C01878=0.000,57.118,70.285,-147.5034,-0.0009,0.0000
C01879=0.000,55.957,72.154,-148.8002,-0.0009,0.0000
C01880=1.768,55.936,72.129,-148.8075,-1.3174,0.0000
C01881=4.219,55.892,72.166,-149.9044,3.8027,0.0000
C01882=7.293,56.844,73.015,-167.6227,12.5357,0.0000
C01883=8.627,60.270,75.143,179.6232,-2.0390,0.0000
C01884=9.417,65.995,78.036,179.4118,-3.7953,0.0000
C01885=10.308,73.408,80.927,179.3669,-4.3506,0.0000
C01886=11.295,81.446,83.062,179.3315,-4.6371,0.0000
C01887=12.427,88.723,84.088,178.6153,-4.2623,0.0000
C01888=15.989,94.030,84.621,177.8322,-1.8057,0.0000
C01889=21.612,96.617,85.050,178.6701,-0.2203,0.0000
C01890=28.131,95.953,85.481,179.9155,0.0246,0.0000
C01891=34.883,93.717,85.762,179.9905,0.0035,0.0000
C01892=41.602,90.934,85.762,179.9908,0.0042,0.0000
C01893=47.957,87.741,85.481,179.9228,0.0423,0.0000
C01894=53.037,83.601,85.050,179.2153,1.0961,0.0000
C01895=55.184,77.795,84.621,179.7437,2.8086,0.0000
C01896=53.949,71.524,84.088,-177.9607,3.9923,0.0000
C01897=49.604,65.578,83.062,-177.1889,3.7534,0.0000
C01898=44.618,59.196,80.927,-177.3673,3.5255,0.0000
C01899=40.007,53.324,78.036,-177.7295,3.1005,0.0000
C01900=36.517,48.718,75.143,-178.8242,1.7083,0.0000
C01901=35.037,45.351,73.015,179.8825,-17.3486,0.0000
C01902=36.538,42.505,72.166,-160.0580,-24.5520,0.0000
C01903=38.303,40.803,72.129,-156.0408,-22.3844,0.0000
C01904=39.567,39.567,72.154,-156.8171,-23.1818,0.0000
C01905=40.803,38.303,72.129,-157.6162,-23.9597,0.0000
C01906=42.506,36.538,72.166,-155.4471,-19.9396,0.0000
C01907=45.352,35.037,73.015,-162.6519,0.1179,0.0000
C01908=48.718,36.517,75.143,178.2917,-1.1758,0.0000
C01909=53.324,40.007,78.036,176.8995,-2.2705,0.0000
C01910=59.196,44.618,80.927,176.4745,-2.6327,0.0000
C01911=65.578,49.604,83.062,176.2466,-2.8111,0.0000
C01912=71.524,53.949,84.088,176.0077,-2.0393,0.0000
C01913=77.795,55.184,84.621,177.1914,0.2563,0.0000
C01914=83.601,53.037,85.050,178.9039,0.7847,0.0000
C01915=87.741,47.957,85.481,179.9577,0.0772,0.0000
C01916=90.934,41.602,85.762,179.9958,0.0092,0.0000
C01917=93.717,34.883,85.762,179.9965,0.0095,0.0000
C01918=95.953,28.131,85.481,179.9754,0.0845,0.0000
C01919=96.617,21.612,85.050,-179.7797,1.3299,0.0000
C01920=94.030,15.989,84.621,-178.1943,2.1678,0.0000
C01921=88.723,12.427,84.088,-175.7377,1.3847,0.0000
C01922=81.446,11.295,83.062,-175.3629,0.6685,0.0000
C01923=73.408,10.308,80.927,-175.6494,0.6331,0.0000
C01924=65.995,9.417,78.036,-176.2047,0.5882,0.0000
C01925=60.270,8.627,75.143,-177.9610,0.3768,0.0000
C01926=56.844,7.293,73.015,167.4643,-12.3773,0.0000
C01927=55.892,4.219,72.166,176.1973,-30.0956,0.0000
C01928=55.936,1.768,72.129,-178.6826,-31.1925,0.0000
C01929=55.957,0.000,72.154,-179.9991,-31.1998,0.0000
C01930=55.936,-1.767,72.129,178.6816,-31.1926,0.0000
C01931=55.892,-4.220,72.166,-176.1946,-30.0948,0.0000
C01932=56.844,-7.293,73.015,-167.4645,-12.3766,0.0000
C01933=60.270,-8.627,75.143,177.9610,0.3768,0.0000
C01934=65.995,-9.417,78.036,176.2047,0.5882,0.0000
C01935=73.408,-10.308,80.927,175.6494,0.6331,0.0000
C01936=81.446,-11.295,83.062,175.3629,0.6685,0.0000
C01937=88.723,-12.427,84.088,175.7377,1.3847,0.0000
C01938=94.030,-15.989,84.621,178.1943,2.1678,0.0000
C01939=96.617,-21.612,85.050,179.7797,1.3299,0.0000
C01940=95.953,-28.131,85.481,-179.9754,0.0845,0.0000
C01941=93.717,-34.883,85.762,-179.9965,0.0095,0.0000
C01942=90.934,-41.602,85.762,-179.9958,0.0092,0.0000
C01943=87.741,-47.957,85.481,-179.9577,0.0772,0.0000
C01944=83.601,-53.037,85.050,-178.9039,0.7847,0.0000
C01945=77.795,-55.184,84.621,-177.1914,0.2563,0.0000
C01946=71.524,-53.949,84.088,-176.0077,-2.0393,0.0000
C01947=65.578,-49.604,83.062,-176.2466,-2.8111,0.0000
C01948=59.196,-44.618,80.927,-176.4745,-2.6327,0.0000
C01949=53.324,-40.007,78.036,-176.8995,-2.2705,0.0000
C01950=48.718,-36.517,75.143,-178.2917,-1.1758,0.0000
C01951=45.351,-35.037,73.015,162.6514,0.1175,0.0000
C01952=42.505,-36.538,72.166,155.4480,-19.9420,0.0000
C01953=40.803,-38.303,72.129,157.6156,-23.9592,0.0000
C01954=39.567,-39.567,72.154,156.8182,-23.1829,0.0000
C01955=38.303,-40.803,72.129,156.0403,-22.3838,0.0000
C01956=36.538,-42.506,72.166,160.0604,-24.5529,0.0000
C01957=35.037,-45.352,73.015,-179.8821,-17.3481,0.0000
C01958=36.517,-48.718,75.143,178.8242,1.7083,0.0000
C01959=40.007,-53.324,78.036,177.7295,3.1005,0.0000
C01960=44.618,-59.196,80.927,177.3673,3.5255,0.0000
C01961=49.604,-65.578,83.062,177.1889,3.7534,0.0000
C01962=53.949,-71.524,84.088,177.9607,3.9923,0.0000
C01963=55.184,-77.795,84.621,-179.7437,2.8086,0.0000
C01964=53.037,-83.601,85.050,-179.2153,1.0961,0.0000
C01965=47.957,-87.741,85.481,-179.9228,0.0423,0.0000
C01966=41.602,-90.934,85.762,-179.9908,0.0042,0.0000
C01967=34.883,-93.717,85.762,-179.9905,0.0035,0.0000
C01968=28.131,-95.953,85.481,-179.9155,0.0246,0.0000
C01969=21.612,-96.617,85.050,-178.6701,-0.2203,0.0000
C01970=15.989,-94.030,84.621,-177.8322,-1.8057,0.0000
C01971=12.427,-88.723,84.088,-178.6153,-4.2623,0.0000
C01972=11.295,-81.446,83.062,-179.3315,-4.6371,0.0000
C01973=10.308,-73.408,80.927,-179.3669,-4.3506,0.0000
C01974=9.417,-65.995,78.036,-179.4118,-3.7953,0.0000
C01975=8.627,-60.270,75.143,-179.6232,-2.0390,0.0000
C01976=7.293,-56.844,73.015,167.6227,12.5357,0.0000
C01977=4.219,-55.892,72.166,149.9044,3.8027,0.0000
C01978=1.768,-55.936,72.129,148.8075,-1.3174,0.0000
C01979=0.000,-55.957,72.154,148.8002,-0.0009,0.0000
C01980=0.000,-55.957,72.154,148.8002,-0.0009,0.0000
C01981=-1.767,-55.936,72.129,148.8074,1.3184,0.0000
C01982=-4.220,-55.892,72.166,149.9052,-3.8054,0.0000
C01983=-7.293,-56.844,73.015,167.6234,-12.5355,0.0000
C01984=-8.627,-60.270,75.143,-179.6232,2.0390,0.0000
C01985=-9.417,-65.995,78.036,-179.4118,3.7953,0.0000
C01986=-10.308,-73.408,80.927,-179.3669,4.3506,0.0000
C01987=-11.295,-81.446,83.062,-179.3315,4.6371,0.0000
C01988=-12.427,-88.723,84.088,-178.6153,4.2623,0.0000
C01989=-15.989,-94.030,84.621,-177.8322,1.8057,0.0000
C01990=-21.612,-96.617,85.050,-178.6701,0.2203,0.0000
C01991=-28.131,-95.953,85.481,-179.9155,-0.0246,0.0000
C01992=-34.883,-93.717,85.762,-179.9905,-0.0035,0.0000
C01993=-41.602,-90.934,85.762,-179.9908,-0.0042,0.0000
C01994=-47.957,-87.741,85.481,-179.9228,-0.0423,0.0000
C01995=-53.037,-83.601,85.050,-179.2153,-1.0961,0.0000
C01996=-55.184,-77.795,84.621,-179.7437,-2.8086,0.0000
C01997=-53.949,-71.524,84.088,177.9607,-3.9923,0.0000
C01998=-49.604,-65.578,83.062,177.1889,-3.7534,0.0000
C01999=-44.618,-59.196,80.927,177.3673,-3.5255,0.0000
///TOOL 0
///POSTYPE ANGLE
///ANGLE
EC00000=-104.1038,0.0000
EC00001=-101.5206,0.0000
EC00002=-99.9757,0.0000
EC00003=-99.7146,0.0000
EC00004=-99.6525,0.0000
EC00005=-99.5501,0.0000
EC00006=-99.1897,0.0000
EC00007=-97.9963,0.0000
EC00008=-95.1629,0.0000
EC00009=-92.4517,0.0000
EC00010=-90.0000,0.0000
EC00011=-87.5483,0.0000
EC00012=-84.8371,0.0000
EC00013=-82.0037,0.0000
EC00014=-80.8103,0.0000
EC00015=-80.4499,0.0000
EC00016=-80.3475,0.0000
EC00017=-80.2854,0.0000
EC00018=-80.0243,0.0000
EC00019=-78.4794,0.0000
EC00020=-75.8962,0.0000
EC00021=-72.7026,0.0000
EC00022=-69.2567,0.0000
EC00023=-65.7434,0.0000
EC00024=-62.2974,0.0000
EC00025=-59.1038,0.0000
EC00026=-56.5207,0.0000
EC00027=-54.9755,0.0000
EC00028=-54.7145,0.0000
EC00029=-54.6524,0.0000
EC00030=-54.5505,0.0000
EC00031=-54.1895,0.0000
EC00032=-52.9962,0.0000
EC00033=-50.1628,0.0000
EC00034=-47.4518,0.0000
EC00035=-45.0000,0.0000
EC00036=-42.5482,0.0000
EC00037=-39.8372,0.0000
EC00038=-37.0034,0.0000
EC00039=-35.8105,0.0000
EC00040=-35.4495,0.0000
EC00041=-35.3476,0.0000
EC00042=-35.2855,0.0000
EC00043=-35.0245,0.0000
EC00044=-33.4793,0.0000
EC00045=-30.8962,0.0000
EC00046=-27.7026,0.0000
EC00047=-24.2566,0.0000
EC00048=-20.7433,0.0000
EC00049=-17.2974,0.0000
EC00050=-14.1038,0.0000
EC00051=-11.5206,0.0000
EC00052=-9.9757,0.0000
EC00053=-9.7146,0.0000
EC00054=-9.6525,0.0000
EC00055=-9.5501,0.0000
EC00056=-9.1897,0.0000
EC00057=-7.9963,0.0000
EC00058=-5.1629,0.0000
EC00059=-2.4517,0.0000
EC00060=0.0000,0.0000
EC00061=0.0000,0.0000
EC00062=2.3954,0.0000
EC00063=5.0881,0.0000
EC00064=7.9350,0.0000
EC00065=9.0911,0.0000
EC00066=9.4060,0.0000
EC00067=9.4709,0.0000
EC00068=9.5004,0.0000
EC00069=9.7298,0.0000
EC00070=11.2851,0.0000
EC00071=13.9122,0.0000
EC00072=17.1736,0.0000
EC00073=20.7008,0.0000
EC00074=24.2992,0.0000
EC00075=27.8267,0.0000
EC00076=31.0877,0.0000
EC00077=33.7152,0.0000
EC00078=35.2699,0.0000
EC00079=35.4993,0.0000
EC00080=35.5293,0.0000
EC00081=35.5938,0.0000
EC00082=35.9087,0.0000
EC00083=37.0654,0.0000
EC00084=39.9123,0.0000
EC00085=42.6047,0.0000
EC00086=45.0000,0.0000
EC00087=47.3953,0.0000
EC00088=50.0883,0.0000
EC00089=52.9346,0.0000
EC00090=54.0913,0.0000
EC00091=54.4062,0.0000
EC00092=54.4707,0.0000
EC00093=54.5007,0.0000
EC00094=54.7301,0.0000
EC00095=56.2848,0.0000
EC00096=58.9123,0.0000
EC00097=62.1733,0.0000
EC00098=65.7008,0.0000
EC00099=69.2992,0.0000
EC00100=72.8264,0.0000
EC00101=76.0878,0.0000
EC00102=78.7149,0.0000
EC00103=80.2702,0.0000
EC00104=80.4996,0.0000
EC00105=80.5291,0.0000
EC00106=80.5940,0.0000
EC00107=80.9089,0.0000
EC00108=82.0650,0.0000
EC00109=84.9119,0.0000
EC00110=87.6046,0.0000
EC00111=90.0000,0.0000
EC00112=92.3954,0.0000
EC00113=95.0881,0.0000
EC00114=97.9350,0.0000
EC00115=99.0911,0.0000
EC00116=99.4060,0.0000
EC00117=99.4709,0.0000
EC00118=99.5004,0.0000
EC00119=99.7298,0.0000
EC00120=101.2851,0.0000
EC00121=103.9122,0.0000
EC00122=107.1736,0.0000
EC00123=110.7008,0.0000
EC00124=114.2992,0.0000
EC00125=117.8267,0.0000
EC00126=121.0877,0.0000
EC00127=123.7152,0.0000
EC00128=125.2699,0.0000
EC00129=125.4993,0.0000
EC00130=125.5293,0.0000
EC00131=125.5938,0.0000
EC00132=125.9087,0.0000
EC00133=127.0654,0.0000
EC00134=129.9123,0.0000
EC00135=132.6047,0.0000
EC00136=135.0000,0.0000
EC00137=137.3953,0.0000
EC00138=140.0883,0.0000
EC00139=142.9346,0.0000
EC00140=144.0913,0.0000
EC00141=144.4062,0.0000
EC00142=144.4707,0.0000
EC00143=144.5007,0.0000
EC00144=144.7301,0.0000
EC00145=146.2848,0.0000
EC00146=148.9123,0.0000
EC00147=152.1733,0.0000
EC00148=155.7008,0.0000
EC00149=159.2992,0.0000
EC00150=162.8264,0.0000
EC00151=166.0878,0.0000
EC00152=168.7149,0.0000
EC00153=170.2702,0.0000
EC00154=170.4996,0.0000
EC00155=170.5291,0.0000
EC00156=170.5940,0.0000
EC00157=170.9089,0.0000
EC00158=172.0650,0.0000
EC00159=174.9119,0.0000
EC00160=177.6046,0.0000
EC00161=180.0000,0.0000
EC00162=180.0000,0.0000
EC00163=-177.6046,0.0000
EC00164=-174.9119,0.0000
EC00165=-172.0650,0.0000
EC00166=-170.9089,0.0000
EC00167=-170.5940,0.0000
EC00168=-170.5291,0.0000
EC00169=-170.4996,0.0000
EC00170=-170.2702,0.0000
EC00171=-168.7149,0.0000
EC00172=-166.0878,0.0000
EC00173=-162.8264,0.0000
EC00174=-159.2992,0.0000
EC00175=-155.7008,0.0000
EC00176=-152.1733,0.0000
EC00177=-148.9123,0.0000
EC00178=-146.2848,0.0000
EC00179=-144.7301,0.0000
EC00180=-144.5007,0.0000
EC00181=-144.4707,0.0000
EC00182=-144.4062,0.0000
EC00183=-144.0913,0.0000
EC00184=-142.9346,0.0000
EC00185=-140.0877,0.0000
EC00186=-137.3953,0.0000
EC00187=-135.0000,0.0000
EC00188=-132.6047,0.0000
EC00189=-129.9117,0.0000
EC00190=-127.0654,0.0000
EC00191=-125.9087,0.0000
EC00192=-125.5938,0.0000
EC00193=-125.5293,0.0000
EC00194=-125.4993,0.0000
EC00195=-125.2699,0.0000
EC00196=-123.7152,0.0000
EC00197=-121.0877,0.0000
EC00198=-117.8267,0.0000
EC00199=-114.2992,0.0000
EC00200=-110.7008,0.0000
EC00201=-107.1736,0.0000
EC00202=-103.9122,0.0000
EC00203=-101.2851,0.0000
EC00204=-99.7298,0.0000
EC00205=-99.5004,0.0000
EC00206=-99.4709,0.0000
EC00207=-99.4060,0.0000
EC00208=-99.0911,0.0000
EC00209=-97.9350,0.0000
EC00210=-95.0881,0.0000
EC00211=-92.3954,0.0000
EC00212=-90.0000,0.0000
EC00213=-87.6046,0.0000
EC00214=-84.9119,0.0000
EC00215=-82.0650,0.0000
EC00216=-80.9089,0.0000
EC00217=-80.5940,0.0000
EC00218=-80.5291,0.0000
EC00219=-80.4996,0.0000
EC00220=-80.2702,0.0000
EC00221=-78.7149,0.0000
EC00222=-76.0878,0.0000
EC00223=-72.8264,0.0000
EC00224=-69.2992,0.0000
EC00225=-65.7008,0.0000
EC00226=-62.1733,0.0000
EC00227=-58.9123,0.0000
EC00228=-56.2848,0.0000
EC00229=-54.7301,0.0000
EC00230=-54.5007,0.0000
EC00231=-54.4707,0.0000
EC00232=-54.4062,0.0000
EC00233=-54.0913,0.0000
EC00234=-52.9346,0.0000
EC00235=-50.0877,0.0000
EC00236=-47.3953,0.0000
EC00237=-45.0000,0.0000
EC00238=-42.6047,0.0000
EC00239=-39.9117,0.0000
EC00240=-37.0654,0.0000
EC00241=-35.9087,0.0000
EC00242=-35.5938,0.0000
EC00243=-35.5293,0.0000
EC00244=-35.4993,0.0000
EC00245=-35.2699,0.0000
EC00246=-33.7152,0.0000
EC00247=-31.0877,0.0000
EC00248=-27.8267,0.0000
EC00249=-24.2992,0.0000
EC00250=-20.7008,0.0000
EC00251=-17.1736,0.0000
EC00252=-13.9122,0.0000
EC00253=-11.2851,0.0000
EC00254=-9.7298,0.0000
EC00255=-9.5004,0.0000
EC00256=-9.4709,0.0000
EC00257=-9.4060,0.0000
EC00258=-9.0911,0.0000
EC00259=-7.9350,0.0000
EC00260=-5.0881,0.0000
EC00261=-2.3954,0.0000
EC00262=0.0000,0.0000
EC00263=0.0000,0.0000
EC00264=2.3363,0.0000
EC00265=5.0104,0.0000
EC00266=7.8714,0.0000
EC00267=8.9912,0.0000
EC00268=9.2604,0.0000
EC00269=9.2892,0.0000
EC00270=9.2905,0.0000
EC00271=9.4907,0.0000
EC00272=11.0568,0.0000
EC00273=13.7273,0.0000
EC00274=17.0541,0.0000
EC00275=20.6599,0.0000
EC00276=24.3400,0.0000
EC00277=27.9461,0.0000
EC00278=31.2727,0.0000
EC00279=33.9430,0.0000
EC00280=35.5096,0.0000
EC00281=35.7099,0.0000
EC00282=35.7103,0.0000
EC00283=35.7399,0.0000
EC00284=36.0092,0.0000
EC00285=37.1289,0.0000
EC00286=39.9895,0.0000
EC00287=42.6632,0.0000
EC00288=45.0000,0.0000
EC00289=47.3362,0.0000
EC00290=50.0105,0.0000
EC00291=52.8711,0.0000
EC00292=53.9908,0.0000
EC00293=54.2601,0.0000
EC00294=54.2897,0.0000
EC00295=54.2901,0.0000
EC00296=54.4904,0.0000
EC00297=56.0570,0.0000
EC00298=58.7273,0.0000
EC00299=62.0539,0.0000
EC00300=65.6600,0.0000
EC00301=69.3401,0.0000
EC00302=72.9459,0.0000
EC00303=76.2727,0.0000
EC00304=78.9432,0.0000
EC00305=80.5093,0.0000
EC00306=80.7095,0.0000
EC00307=80.7108,0.0000
EC00308=80.7396,0.0000
EC00309=81.0088,0.0000
EC00310=82.1286,0.0000
EC00311=84.9896,0.0000
EC00312=87.6637,0.0000
EC00313=90.0000,0.0000
EC00314=92.3363,0.0000
EC00315=95.0112,0.0000
EC00316=97.8714,0.0000
EC00317=98.9912,0.0000
EC00318=99.2604,0.0000
EC00319=99.2892,0.0000
EC00320=99.2905,0.0000
EC00321=99.4907,0.0000
EC00322=101.0568,0.0000
EC00323=103.7273,0.0000
EC00324=107.0541,0.0000
EC00325=110.6599,0.0000
EC00326=114.3400,0.0000
EC00327=117.9461,0.0000
EC00328=121.2727,0.0000
EC00329=123.9430,0.0000
EC00330=125.5096,0.0000
EC00331=125.7099,0.0000
EC00332=125.7103,0.0000
EC00333=125.7399,0.0000
EC00334=126.0092,0.0000
EC00335=127.1289,0.0000
EC00336=129.9895,0.0000
EC00337=132.6632,0.0000
EC00338=135.0000,0.0000
EC00339=137.3362,0.0000
EC00340=140.0105,0.0000
EC00341=142.8711,0.0000
EC00342=143.9908,0.0000
EC00343=144.2601,0.0000
EC00344=144.2897,0.0000
EC00345=144.2901,0.0000
EC00346=144.4904,0.0000
EC00347=146.0570,0.0000
EC00348=148.7273,0.0000
EC00349=152.0539,0.0000
EC00350=155.6600,0.0000
EC00351=159.3401,0.0000
EC00352=162.9459,0.0000
EC00353=166.2727,0.0000
EC00354=168.9432,0.0000
EC00355=170.5093,0.0000
EC00356=170.7095,0.0000
EC00357=170.7108,0.0000
EC00358=170.7396,0.0000
EC00359=171.0088,0.0000
EC00360=172.1286,0.0000
EC00361=174.9896,0.0000
EC00362=177.6637,0.0000
EC00363=180.0000,0.0000
EC00364=180.0000,0.0000
EC00365=-177.6637,0.0000
EC00366=-174.9888,0.0000
EC00367=-172.1286,0.0000
EC00368=-171.0088,0.0000
EC00369=-170.7396,0.0000
EC00370=-170.7108,0.0000
EC00371=-170.7095,0.0000
EC00372=-170.5093,0.0000
EC00373=-168.9432,0.0000
EC00374=-166.2727,0.0000
EC00375=-162.9459,0.0000
EC00376=-159.3401,0.0000
EC00377=-155.6600,0.0000
EC00378=-152.0539,0.0000
EC00379=-148.7273,0.0000
EC00380=-146.0570,0.0000
EC00381=-144.4904,0.0000
EC00382=-144.2901,0.0000
EC00383=-144.2897,0.0000
EC00384=-144.2601,0.0000
EC00385=-143.9908,0.0000
EC00386=-142.8711,0.0000
EC00387=-140.0105,0.0000
EC00388=-137.3368,0.0000
EC00389=-135.0000,0.0000
EC00390=-132.6638,0.0000
EC00391=-129.9895,0.0000
EC00392=-127.1289,0.0000
EC00393=-126.0092,0.0000
EC00394=-125.7399,0.0000
EC00395=-125.7103,0.0000
EC00396=-125.7099,0.0000
EC00397=-125.5096,0.0000
EC00398=-123.9430,0.0000
EC00399=-121.2727,0.0000
EC00400=-117.9461,0.0000
EC00401=-114.3400,0.0000
EC00402=-110.6599,0.0000
EC00403=-107.0541,0.0000
EC00404=-103.7273,0.0000
EC00405=-101.0568,0.0000
EC00406=-99.4907,0.0000
EC00407=-99.2905,0.0000
EC00408=-99.2892,0.0000
EC00409=-99.2604,0.0000
EC00410=-98.9912,0.0000
EC00411=-97.8714,0.0000
EC00412=-95.0104,0.0000
EC00413=-92.3363,0.0000
EC00414=-90.0000,0.0000
EC00415=-87.6637,0.0000
EC00416=-84.9888,0.0000
EC00417=-82.1286,0.0000
EC00418=-81.0088,0.0000
EC00419=-80.7396,0.0000
EC00420=-80.7108,0.0000
EC00421=-80.7095,0.0000
EC00422=-80.5093,0.0000
EC00423=-78.9432,0.0000
EC00424=-76.2727,0.0000
EC00425=-72.9459,0.0000
EC00426=-69.3401,0.0000
EC00427=-65.6600,0.0000
EC00428=-62.0539,0.0000
EC00429=-58.7273,0.0000
EC00430=-56.0570,0.0000
EC00431=-54.4904,0.0000
EC00432=-54.2901,0.0000
EC00433=-54.2897,0.0000
EC00434=-54.2601,0.0000
EC00435=-53.9908,0.0000
EC00436=-52.8711,0.0000
EC00437=-50.0105,0.0000
EC00438=-47.3368,0.0000
EC00439=-45.0000,0.0000
EC00440=-42.6638,0.0000
EC00441=-39.9895,0.0000
EC00442=-37.1289,0.0000
EC00443=-36.0092,0.0000
EC00444=-35.7399,0.0000
EC00445=-35.7103,0.0000
EC00446=-35.7099,0.0000
EC00447=-35.5096,0.0000
EC00448=-33.9430,0.0000
EC00449=-31.2727,0.0000
EC00450=-27.9461,0.0000
EC00451=-24.3400,0.0000
EC00452=-20.6599,0.0000
EC00453=-17.0541,0.0000
EC00454=-13.7273,0.0000
EC00455=-11.0568,0.0000
EC00456=-9.4907,0.0000
EC00457=-9.2905,0.0000
EC00458=-9.2892,0.0000
EC00459=-9.2604,0.0000
EC00460=-8.9912,0.0000
EC00461=-7.8714,0.0000
EC00462=-5.0112,0.0000
EC00463=-2.3363,0.0000
EC00464=0.0000,0.0000
EC00465=0.0000,0.0000
EC00466=2.2761,0.0000
EC00467=4.9310,0.0000
EC00468=7.8063,0.0000
EC00469=8.8881,0.0000
EC00470=9.1126,0.0000
EC00471=9.1102,0.0000
EC00472=9.0849,0.0000
EC00473=9.2589,0.0000
EC00474=10.8371,0.0000
EC00475=13.5503,0.0000
EC00476=16.9400,0.0000
EC00477=20.6205,0.0000
EC00478=24.3795,0.0000
EC00479=28.0601,0.0000
EC00480=31.4498,0.0000
EC00481=34.1627,0.0000
EC00482=35.7411,0.0000
EC00483=35.9150,0.0000
EC00484=35.8901,0.0000
EC00485=35.8871,0.0000
EC00486=36.1114,0.0000
EC00487=37.1942,0.0000
EC00488=40.0690,0.0000
EC00489=42.7235,0.0000
EC00490=45.0000,0.0000
EC00491=47.2759,0.0000
EC00492=49.9310,0.0000
EC00493=52.8058,0.0000
EC00494=53.8886,0.0000
EC00495=54.1129,0.0000
EC00496=54.1099,0.0000
EC00497=54.0850,0.0000
EC00498=54.2589,0.0000
EC00499=55.8373,0.0000
EC00500=58.5502,0.0000
EC00501=61.9399,0.0000
EC00502=65.6205,0.0000
EC00503=69.3795,0.0000
EC00504=73.0600,0.0000
EC00505=76.4497,0.0000
EC00506=79.1629,0.0000
EC00507=80.7411,0.0000
EC00508=80.9151,0.0000
EC00509=80.8898,0.0000
EC00510=80.8874,0.0000
EC00511=81.1119,0.0000
EC00512=82.1937,0.0000
EC00513=85.0690,0.0000
EC00514=87.7239,0.0000
EC00515=90.0000,0.0000
EC00516=92.2761,0.0000
EC00517=94.9310,0.0000
EC00518=97.8063,0.0000
EC00519=98.8881,0.0000
EC00520=99.1126,0.0000
EC00521=99.1102,0.0000
EC00522=99.0849,0.0000
EC00523=99.2589,0.0000
EC00524=100.8371,0.0000
EC00525=103.5503,0.0000
EC00526=106.9400,0.0000
EC00527=110.6205,0.0000
EC00528=114.3795,0.0000
EC00529=118.0601,0.0000
EC00530=121.4498,0.0000
EC00531=124.1627,0.0000
EC00532=125.7411,0.0000
EC00533=125.9150,0.0000
EC00534=125.8901,0.0000
EC00535=125.8871,0.0000
EC00536=126.1114,0.0000
EC00537=127.1942,0.0000
EC00538=130.0690,0.0000
EC00539=132.7235,0.0000
EC00540=135.0000,0.0000
EC00541=137.2759,0.0000
EC00542=139.9310,0.0000
EC00543=142.8058,0.0000
EC00544=143.8886,0.0000
EC00545=144.1129,0.0000
EC00546=144.1099,0.0000
EC00547=144.0850,0.0000
EC00548=144.2589,0.0000
EC00549=145.8373,0.0000
EC00550=148.5502,0.0000
EC00551=151.9399,0.0000
EC00552=155.6205,0.0000
EC00553=159.3795,0.0000
EC00554=163.0600,0.0000
EC00555=166.4497,0.0000
EC00556=169.1629,0.0000
EC00557=170.7411,0.0000
EC00558=170.9151,0.0000
EC00559=170.8898,0.0000
EC00560=170.8874,0.0000
EC00561=171.1119,0.0000
EC00562=172.1937,0.0000
EC00563=175.0690,0.0000
EC00564=177.7239,0.0000
EC00565=180.0000,0.0000
EC00566=180.0000,0.0000
EC00567=-177.7239,0.0000
EC00568=-175.0690,0.0000
EC00569=-172.1937,0.0000
EC00570=-171.1119,0.0000
EC00571=-170.8874,0.0000
EC00572=-170.8898,0.0000
EC00573=-170.9151,0.0000
EC00574=-170.7411,0.0000
EC00575=-169.1629,0.0000
EC00576=-166.4497,0.0000
EC00577=-163.0600,0.0000
EC00578=-159.3795,0.0000
EC00579=-155.6205,0.0000
EC00580=-151.9399,0.0000
EC00581=-148.5502,0.0000
EC00582=-145.8373,0.0000
EC00583=-144.2589,0.0000
EC00584=-144.0850,0.0000
EC00585=-144.1099,0.0000
EC00586=-144.1129,0.0000
EC00587=-143.8886,0.0000
EC00588=-142.8058,0.0000
EC00589=-139.9310,0.0000
EC00590=-137.2765,0.0000
EC00591=-135.0000,0.0000
EC00592=-132.7241,0.0000
EC00593=-130.0690,0.0000
EC00594=-127.1942,0.0000
EC00595=-126.1114,0.0000
EC00596=-125.8871,0.0000
EC00597=-125.8901,0.0000
EC00598=-125.9150,0.0000
EC00599=-125.7411,0.0000
EC00600=-124.1627,0.0000
EC00601=-121.4498,0.0000
EC00602=-118.0601,0.0000
EC00603=-114.3795,0.0000
EC00604=-110.6205,0.0000
EC00605=-106.9400,0.0000
EC00606=-103.5503,0.0000
EC00607=-100.8371,0.0000
EC00608=-99.2589,0.0000
EC00609=-99.0849,0.0000
EC00610=-99.1102,0.0000
EC00611=-99.1126,0.0000
EC00612=-98.8881,0.0000
EC00613=-97.8063,0.0000
EC00614=-94.9310,0.0000
EC00615=-92.2761,0.0000
EC00616=-90.0000,0.0000
EC00617=-87.7239,0.0000
EC00618=-85.0690,0.0000
EC00619=-82.1937,0.0000
EC00620=-81.1119,0.0000
EC00621=-80.8874,0.0000
EC00622=-80.8898,0.0000
EC00623=-80.9151,0.0000
EC00624=-80.7411,0.0000
EC00625=-79.1629,0.0000
EC00626=-76.4497,0.0000
EC00627=-73.0600,0.0000
EC00628=-69.3795,0.0000
EC00629=-65.6205,0.0000
EC00630=-61.9399,0.0000
EC00631=-58.5502,0.0000
EC00632=-55.8373,0.0000
EC00633=-54.2589,0.0000
EC00634=-54.0850,0.0000
EC00635=-54.1099,0.0000
EC00636=-54.1129,0.0000
EC00637=-53.8886,0.0000
EC00638=-52.8058,0.0000
EC00639=-49.9310,0.0000
EC00640=-47.2765,0.0000
EC00641=-45.0000,0.0000
EC00642=-42.7241,0.0000
EC00643=-40.0690,0.0000
EC00644=-37.1942,0.0000
EC00645=-36.1114,0.0000
EC00646=-35.8871,0.0000
EC00647=-35.8901,0.0000
EC00648=-35.9150,0.0000
EC00649=-35.7411,0.0000
EC00650=-34.1627,0.0000
EC00651=-31.4498,0.0000
EC00652=-28.0601,0.0000
EC00653=-24.3795,0.0000
EC00654=-20.6205,0.0000
EC00655=-16.9400,0.0000
EC00656=-13.5503,0.0000
EC00657=-10.8371,0.0000
EC00658=-9.2589,0.0000
EC00659=-9.0849,0.0000
EC00660=-9.1102,0.0000
EC00661=-9.1126,0.0000
EC00662=-8.8881,0.0000
EC00663=-7.8063,0.0000
EC00664=-4.9310,0.0000
EC00665=-2.2761,0.0000
EC00666=0.0000,0.0000
EC00667=0.0000,0.0000
EC00668=2.2137,0.0000
EC00669=4.8488,0.0000
EC00670=7.7390,0.0000
EC00671=8.7837,0.0000
EC00672=8.9651,0.0000
EC00673=8.9329,0.0000
EC00674=8.8862,0.0000
EC00675=9.0366,0.0000
EC00676=10.6278,0.0000
EC00677=13.3823,0.0000
EC00678=16.8314,0.0000
EC00679=20.5837,0.0000
EC00680=24.4165,0.0000
EC00681=28.1685,0.0000
EC00682=31.6178,0.0000
EC00683=34.3719,0.0000
EC00684=35.9638,0.0000
EC00685=36.1137,0.0000
EC00686=36.0668,0.0000
EC00687=36.0347,0.0000
EC00688=36.2163,0.0000
EC00689=37.2611,0.0000
EC00690=40.1513,0.0000
EC00691=42.7862,0.0000
EC00692=45.0000,0.0000
EC00693=47.2138,0.0000
EC00694=49.8487,0.0000
EC00695=52.7389,0.0000
EC00696=53.7837,0.0000
EC00697=53.9653,0.0000
EC00698=53.9332,0.0000
EC00699=53.8863,0.0000
EC00700=54.0362,0.0000
EC00701=55.6281,0.0000
EC00702=58.3822,0.0000
EC00703=61.8315,0.0000
EC00704=65.5835,0.0000
EC00705=69.4163,0.0000
EC00706=73.1686,0.0000
EC00707=76.6177,0.0000
EC00708=79.3722,0.0000
EC00709=80.9634,0.0000
EC00710=81.1138,0.0000
EC00711=81.0671,0.0000
EC00712=81.0349,0.0000
EC00713=81.2163,0.0000
EC00714=82.2610,0.0000
EC00715=85.1512,0.0000
EC00716=87.7863,0.0000
EC00717=90.0000,0.0000
EC00718=92.2137,0.0000
EC00719=94.8488,0.0000
EC00720=97.7390,0.0000
EC00721=98.7837,0.0000
EC00722=98.9651,0.0000
EC00723=98.9329,0.0000
EC00724=98.8862,0.0000
EC00725=99.0366,0.0000
EC00726=100.6278,0.0000
EC00727=103.3823,0.0000
EC00728=106.8314,0.0000
EC00729=110.5837,0.0000
EC00730=114.4165,0.0000
EC00731=118.1685,0.0000
EC00732=121.6178,0.0000
EC00733=124.3719,0.0000
EC00734=125.9638,0.0000
EC00735=126.1137,0.0000
EC00736=126.0668,0.0000
EC00737=126.0347,0.0000
EC00738=126.2163,0.0000
EC00739=127.2611,0.0000
EC00740=130.1513,0.0000
EC00741=132.7862,0.0000
EC00742=135.0000,0.0000
EC00743=137.2138,0.0000
EC00744=139.8487,0.0000
EC00745=142.7389,0.0000
EC00746=143.7837,0.0000
EC00747=143.9653,0.0000
EC00748=143.9332,0.0000
EC00749=143.8863,0.0000
EC00750=144.0362,0.0000
EC00751=145.6281,0.0000
EC00752=148.3822,0.0000
EC00753=151.8315,0.0000
EC00754=155.5835,0.0000
EC00755=159.4163,0.0000
EC00756=163.1686,0.0000
EC00757=166.6177,0.0000
EC00758=169.3722,0.0000
EC00759=170.9634,0.0000
EC00760=171.1138,0.0000
EC00761=171.0671,0.0000
EC00762=171.0349,0.0000
EC00763=171.2163,0.0000
EC00764=172.2610,0.0000
EC00765=175.1512,0.0000
EC00766=177.7863,0.0000
EC00767=180.0000,0.0000
EC00768=180.0000,0.0000
EC00769=-177.7863,0.0000
EC00770=-175.1512,0.0000
EC00771=-172.2610,0.0000
EC00772=-171.2163,0.0000
EC00773=-171.0349,0.0000
EC00774=-171.0671,0.0000
EC00775=-171.1138,0.0000
EC00776=-170.9634,0.0000
EC00777=-169.3722,0.0000
EC00778=-166.6177,0.0000
EC00779=-163.1686,0.0000
EC00780=-159.4163,0.0000
EC00781=-155.5835,0.0000
EC00782=-151.8315,0.0000
EC00783=-148.3822,0.0000
EC00784=-145.6281,0.0000
EC00785=-144.0362,0.0000
EC00786=-143.8863,0.0000
EC00787=-143.9332,0.0000
EC00788=-143.9653,0.0000
EC00789=-143.7837,0.0000
EC00790=-142.7389,0.0000
EC00791=-139.8487,0.0000
EC00792=-137.2138,0.0000
EC00793=-135.0000,0.0000
EC00794=-132.7862,0.0000
EC00795=-130.1513,0.0000
EC00796=-127.2611,0.0000
EC00797=-126.2163,0.0000
EC00798=-126.0347,0.0000
EC00799=-126.0668,0.0000
EC00800=-126.1137,0.0000
EC00801=-125.9638,0.0000
EC00802=-124.3719,0.0000
EC00803=-121.6178,0.0000
EC00804=-118.1685,0.0000
EC00805=-114.4165,0.0000
EC00806=-110.5837,0.0000
EC00807=-106.8314,0.0000
EC00808=-103.3823,0.0000
EC00809=-100.6278,0.0000
EC00810=-99.0366,0.0000
EC00811=-98.8862,0.0000
EC00812=-98.9329,0.0000
EC00813=-98.9651,0.0000
EC00814=-98.7837,0.0000
EC00815=-97.7390,0.0000
EC00816=-94.8488,0.0000
EC00817=-92.2137,0.0000
EC00818=-90.0000,0.0000
EC00819=-87.7863,0.0000
EC00820=-85.1512,0.0000
EC00821=-82.2610,0.0000
EC00822=-81.2163,0.0000
EC00823=-81.0349,0.0000
EC00824=-81.0671,0.0000
EC00825=-81.1138,0.0000
EC00826=-80.9634,0.0000
EC00827=-79.3722,0.0000
EC00828=-76.6177,0.0000
EC00829=-73.1686,0.0000
EC00830=-69.4163,0.0000
EC00831=-65.5835,0.0000
EC00832=-61.8315,0.0000
EC00833=-58.3822,0.0000
EC00834=-55.6281,0.0000
EC00835=-54.0362,0.0000
EC00836=-53.8863,0.0000
EC00837=-53.9332,0.0000
EC00838=-53.9653,0.0000
EC00839=-53.7837,0.0000
EC00840=-52.7389,0.0000
EC00841=-49.8487,0.0000
EC00842=-47.2138,0.0000
EC00843=-45.0000,0.0000
EC00844=-42.7862,0.0000
EC00845=-40.1513,0.0000
EC00846=-37.2611,0.0000
EC00847=-36.2163,0.0000
EC00848=-36.0347,0.0000
EC00849=-36.0668,0.0000
EC00850=-36.1137,0.0000
EC00851=-35.9638,0.0000
EC00852=-34.3719,0.0000
EC00853=-31.6178,0.0000
EC00854=-28.1685,0.0000
EC00855=-24.4165,0.0000
EC00856=-20.5837,0.0000
EC00857=-16.8314,0.0000
EC00858=-13.3823,0.0000
EC00859=-10.6278,0.0000
EC00860=-9.0366,0.0000
EC00861=-8.8862,0.0000
EC00862=-8.9329,0.0000
EC00863=-8.9651,0.0000
EC00864=-8.7837,0.0000
EC00865=-7.7390,0.0000
EC00866=-4.8488,0.0000
EC00867=-2.2137,0.0000
EC00868=0.0000,0.0000
EC00869=0.0000,0.0000
EC00870=2.1497,0.0000
EC00871=4.7644,0.0000
EC00872=7.6702,0.0000
EC00873=8.6786,0.0000
EC00874=8.8182,0.0000
EC00875=8.7594,0.0000
EC00876=8.6938,0.0000
EC00877=8.8243,0.0000
EC00878=10.4296,0.0000
EC00879=13.2238,0.0000
EC00880=16.7302,0.0000
EC00881=20.5487,0.0000
EC00882=24.4516,0.0000
EC00883=28.2700,0.0000
EC00884=31.7764,0.0000
EC00885=34.5698,0.0000
EC00886=36.1755,0.0000
EC00887=36.3059,0.0000
EC00888=36.2401,0.0000
EC00889=36.1817,0.0000
EC00890=36.3218,0.0000
EC00891=37.3300,0.0000
EC00892=40.2352,0.0000
EC00893=42.8504,0.0000
EC00894=45.0000,0.0000
EC00895=47.1496,0.0000
EC00896=49.7648,0.0000
EC00897=52.6700,0.0000
EC00898=53.6782,0.0000
EC00899=53.8183,0.0000
EC00900=53.7599,0.0000
EC00901=53.6941,0.0000
EC00902=53.8245,0.0000
EC00903=55.4302,0.0000
EC00904=58.2236,0.0000
EC00905=61.7300,0.0000
EC00906=65.5484,0.0000
EC00907=69.4513,0.0000
EC00908=73.2698,0.0000
EC00909=76.7762,0.0000
EC00910=79.5704,0.0000
EC00911=81.1757,0.0000
EC00912=81.3062,0.0000
EC00913=81.2406,0.0000
EC00914=81.1818,0.0000
EC00915=81.3214,0.0000
EC00916=82.3298,0.0000
EC00917=85.2356,0.0000
EC00918=87.8503,0.0000
EC00919=90.0000,0.0000
EC00920=92.1497,0.0000
EC00921=94.7644,0.0000
EC00922=97.6701,0.0000
EC00923=98.6786,0.0000
EC00924=98.8182,0.0000
EC00925=98.7594,0.0000
EC00926=98.6938,0.0000
EC00927=98.8243,0.0000
EC00928=100.4296,0.0000
EC00929=103.2238,0.0000
EC00930=106.7302,0.0000
EC00931=110.5487,0.0000
EC00932=114.4516,0.0000
EC00933=118.2700,0.0000
EC00934=121.7764,0.0000
EC00935=124.5698,0.0000
EC00936=126.1755,0.0000
EC00937=126.3059,0.0000
EC00938=126.2401,0.0000
EC00939=126.1817,0.0000
EC00940=126.3218,0.0000
EC00941=127.3300,0.0000
EC00942=130.2352,0.0000
EC00943=132.8504,0.0000
EC00944=135.0000,0.0000
EC00945=137.1496,0.0000
EC00946=139.7648,0.0000
EC00947=142.6700,0.0000
EC00948=143.6782,0.0000
EC00949=143.8183,0.0000
EC00950=143.7599,0.0000
EC00951=143.6941,0.0000
EC00952=143.8245,0.0000
EC00953=145.4302,0.0000
EC00954=148.2236,0.0000
EC00955=151.7300,0.0000
EC00956=155.5484,0.0000
EC00957=159.4513,0.0000
EC00958=163.2698,0.0000
EC00959=166.7762,0.0000
EC00960=169.5704,0.0000
EC00961=171.1757,0.0000
EC00962=171.3062,0.0000
EC00963=171.2406,0.0000
EC00964=171.1818,0.0000
EC00965=171.3214,0.0000
EC00966=172.3298,0.0000
EC00967=175.2356,0.0000
EC00968=177.8503,0.0000
EC00969=180.0000,0.0000
EC00970=180.0000,0.0000
EC00971=-177.8503,0.0000
EC00972=-175.2356,0.0000
EC00973=-172.3299,0.0000
EC00974=-171.3214,0.0000
EC00975=-171.1818,0.0000
EC00976=-171.2406,0.0000
EC00977=-171.3062,0.0000
EC00978=-171.1757,0.0000
EC00979=-169.5704,0.0000
EC00980=-166.7762,0.0000
EC00981=-163.2698,0.0000
EC00982=-159.4513,0.0000
EC00983=-155.5484,0.0000
EC00984=-151.7300,0.0000
EC00985=-148.2236,0.0000
EC00986=-145.4302,0.0000
EC00987=-143.8245,0.0000
EC00988=-143.6941,0.0000
EC00989=-143.7599,0.0000
EC00990=-143.8183,0.0000
EC00991=-143.6782,0.0000
EC00992=-142.6700,0.0000
EC00993=-139.7648,0.0000
EC00994=-137.1496,0.0000
EC00995=-135.0000,0.0000
EC00996=-132.8504,0.0000
EC00997=-130.2352,0.0000
EC00998=-127.3300,0.0000
EC00999=-126.3218,0.0000
EC01000=-126.1817,0.0000
EC01001=-126.2401,0.0000
EC01002=-126.3059,0.0000
EC01003=-126.1755,0.0000
EC01004=-124.5698,0.0000
EC01005=-121.7764,0.0000
EC01006=-118.2700,0.0000
EC01007=-114.4516,0.0000
EC01008=-110.5487,0.0000
EC01009=-106.7302,0.0000
EC01010=-103.2238,0.0000
EC01011=-100.4296,0.0000
EC01012=-98.8243,0.0000
EC01013=-98.6938,0.0000
EC01014=-98.7594,0.0000
EC01015=-98.8182,0.0000
EC01016=-98.6786,0.0000
EC01017=-97.6702,0.0000
EC01018=-94.7644,0.0000
EC01019=-92.1497,0.0000
EC01020=-90.0000,0.0000
EC01021=-87.8503,0.0000
EC01022=-85.2356,0.0000
EC01023=-82.3299,0.0000
EC01024=-81.3214,0.0000
EC01025=-81.1818,0.0000
EC01026=-81.2406,0.0000
EC01027=-81.3062,0.0000
EC01028=-81.1757,0.0000
EC01029=-79.5704,0.0000
EC01030=-76.7762,0.0000
EC01031=-73.2698,0.0000
EC01032=-69.4513,0.0000
EC01033=-65.5484,0.0000
EC01034=-61.7300,0.0000
EC01035=-58.2236,0.0000
EC01036=-55.4302,0.0000
EC01037=-53.8245,0.0000
EC01038=-53.6941,0.0000
EC01039=-53.7599,0.0000
EC01040=-53.8183,0.0000
EC01041=-53.6782,0.0000
EC01042=-52.6700,0.0000
EC01043=-49.7648,0.0000
EC01044=-47.1496,0.0000
EC01045=-45.0000,0.0000
EC01046=-42.8504,0.0000
EC01047=-40.2352,0.0000
EC01048=-37.3300,0.0000
EC01049=-36.3218,0.0000
EC01050=-36.1817,0.0000
EC01051=-36.2401,0.0000
EC01052=-36.3059,0.0000
EC01053=-36.1755,0.0000
EC01054=-34.5698,0.0000
EC01055=-31.7764,0.0000
EC01056=-28.2700,0.0000
EC01057=-24.4516,0.0000
EC01058=-20.5487,0.0000
EC01059=-16.7302,0.0000
EC01060=-13.2238,0.0000
EC01061=-10.4296,0.0000
EC01062=-8.8243,0.0000
EC01063=-8.6938,0.0000
EC01064=-8.7594,0.0000
EC01065=-8.8182,0.0000
EC01066=-8.6786,0.0000
EC01067=-7.6701,0.0000
EC01068=-4.7644,0.0000
EC01069=-2.1497,0.0000
EC01070=0.0000,0.0000
EC01071=0.0000,0.0000
EC01072=2.0841,0.0000
EC01073=4.6784,0.0000
EC01074=7.6002,0.0000
EC01075=8.5715,0.0000
EC01076=8.6723,0.0000
EC01077=8.5913,0.0000
EC01078=8.5111,0.0000
EC01079=8.6248,0.0000
EC01080=10.2442,0.0000
EC01081=13.0758,0.0000
EC01082=16.6354,0.0000
EC01083=20.5162,0.0000
EC01084=24.4836,0.0000
EC01085=28.3648,0.0000
EC01086=31.9242,0.0000
EC01087=34.7559,0.0000
EC01088=36.3755,0.0000
EC01089=36.4893,0.0000
EC01090=36.4090,0.0000
EC01091=36.3280,0.0000
EC01092=36.4285,0.0000
EC01093=37.4001,0.0000
EC01094=40.3225,0.0000
EC01095=42.9160,0.0000
EC01096=45.0000,0.0000
EC01097=47.0840,0.0000
EC01098=49.6788,0.0000
EC01099=52.5999,0.0000
EC01100=53.5715,0.0000
EC01101=53.6720,0.0000
EC01102=53.5910,0.0000
EC01103=53.5107,0.0000
EC01104=53.6245,0.0000
EC01105=55.2441,0.0000
EC01106=58.0758,0.0000
EC01107=61.6352,0.0000
EC01108=65.5164,0.0000
EC01109=69.4838,0.0000
EC01110=73.3646,0.0000
EC01111=76.9242,0.0000
EC01112=79.7558,0.0000
EC01113=81.3752,0.0000
EC01114=81.4889,0.0000
EC01115=81.4087,0.0000
EC01116=81.3277,0.0000
EC01117=81.4285,0.0000
EC01118=82.3998,0.0000
EC01119=85.3216,0.0000
EC01120=87.9159,0.0000
EC01121=90.0000,0.0000
EC01122=92.0841,0.0000
EC01123=94.6784,0.0000
EC01124=97.6002,0.0000
EC01125=98.5715,0.0000
EC01126=98.6723,0.0000
EC01127=98.5913,0.0000
EC01128=98.5111,0.0000
EC01129=98.6248,0.0000
EC01130=100.2442,0.0000
EC01131=103.0758,0.0000
EC01132=106.6354,0.0000
EC01133=110.5162,0.0000
EC01134=114.4836,0.0000
EC01135=118.3648,0.0000
EC01136=121.9242,0.0000
EC01137=124.7559,0.0000
EC01138=126.3755,0.0000
EC01139=126.4893,0.0000
EC01140=126.4090,0.0000
EC01141=126.3280,0.0000
EC01142=126.4285,0.0000
EC01143=127.4001,0.0000
EC01144=130.3225,0.0000
EC01145=132.9160,0.0000
EC01146=135.0000,0.0000
EC01147=137.0840,0.0000
EC01148=139.6788,0.0000
EC01149=142.5999,0.0000
EC01150=143.5715,0.0000
EC01151=143.6720,0.0000
EC01152=143.5910,0.0000
EC01153=143.5107,0.0000
EC01154=143.6245,0.0000
EC01155=145.2441,0.0000
EC01156=148.0758,0.0000
EC01157=151.6352,0.0000
EC01158=155.5164,0.0000
EC01159=159.4838,0.0000
EC01160=163.3646,0.0000
EC01161=166.9242,0.0000
EC01162=169.7558,0.0000
EC01163=171.3752,0.0000
EC01164=171.4889,0.0000
EC01165=171.4087,0.0000
EC01166=171.3277,0.0000
EC01167=171.4285,0.0000
EC01168=172.3998,0.0000
EC01169=175.3216,0.0000
EC01170=177.9159,0.0000
EC01171=180.0000,0.0000
EC01172=180.0000,0.0000
EC01173=-177.9159,0.0000
EC01174=-175.3216,0.0000
EC01175=-172.3998,0.0000
EC01176=-171.4285,0.0000
EC01177=-171.3277,0.0000
EC01178=-171.4087,0.0000
EC01179=-171.4889,0.0000
EC01180=-171.3752,0.0000
EC01181=-169.7558,0.0000
EC01182=-166.9242,0.0000
EC01183=-163.3646,0.0000
EC01184=-159.4838,0.0000
EC01185=-155.5164,0.0000
EC01186=-151.6352,0.0000
EC01187=-148.0758,0.0000
EC01188=-145.2441,0.0000
EC01189=-143.6245,0.0000
EC01190=-143.5107,0.0000
EC01191=-143.5910,0.0000
EC01192=-143.6720,0.0000
EC01193=-143.5715,0.0000
EC01194=-142.5999,0.0000
EC01195=-139.6775,0.0000
EC01196=-137.0840,0.0000
EC01197=-135.0000,0.0000
EC01198=-132.9160,0.0000
EC01199=-130.3212,0.0000
EC01200=-127.4001,0.0000
EC01201=-126.4285,0.0000
EC01202=-126.3280,0.0000
EC01203=-126.4090,0.0000
EC01204=-126.4893,0.0000
EC01205=-126.3755,0.0000
EC01206=-124.7559,0.0000
EC01207=-121.9242,0.0000
EC01208=-118.3648,0.0000
EC01209=-114.4836,0.0000
EC01210=-110.5162,0.0000
EC01211=-106.6354,0.0000
EC01212=-103.0758,0.0000
EC01213=-100.2442,0.0000
EC01214=-98.6248,0.0000
EC01215=-98.5111,0.0000
EC01216=-98.5913,0.0000
EC01217=-98.6723,0.0000
EC01218=-98.5715,0.0000
EC01219=-97.6002,0.0000
EC01220=-94.6784,0.0000
EC01221=-92.0841,0.0000
EC01222=-90.0000,0.0000
EC01223=-87.9159,0.0000
EC01224=-85.3216,0.0000
EC01225=-82.3998,0.0000
EC01226=-81.4285,0.0000
EC01227=-81.3277,0.0000
EC01228=-81.4087,0.0000
EC01229=-81.4889,0.0000
EC01230=-81.3752,0.0000
EC01231=-79.7558,0.0000
EC01232=-76.9242,0.0000
EC01233=-73.3646,0.0000
EC01234=-69.4838,0.0000
EC01235=-65.5164,0.0000
EC01236=-61.6352,0.0000
EC01237=-58.0758,0.0000
EC01238=-55.2441,0.0000
EC01239=-53.6245,0.0000
EC01240=-53.5107,0.0000
EC01241=-53.5910,0.0000
EC01242=-53.6720,0.0000
EC01243=-53.5715,0.0000
EC01244=-52.5999,0.0000
EC01245=-49.6775,0.0000
EC01246=-47.0840,0.0000
EC01247=-45.0000,0.0000
EC01248=-42.9160,0.0000
EC01249=-40.3212,0.0000
EC01250=-37.4001,0.0000
EC01251=-36.4285,0.0000
EC01252=-36.3280,0.0000
EC01253=-36.4090,0.0000
EC01254=-36.4893,0.0000
EC01255=-36.3755,0.0000
EC01256=-34.7559,0.0000
EC01257=-31.9242,0.0000
EC01258=-28.3648,0.0000
EC01259=-24.4836,0.0000
EC01260=-20.5162,0.0000
EC01261=-16.6354,0.0000
EC01262=-13.0758,0.0000
EC01263=-10.2442,0.0000
EC01264=-8.6248,0.0000
EC01265=-8.5111,0.0000
EC01266=-8.5913,0.0000
EC01267=-8.6723,0.0000
EC01268=-8.5715,0.0000
EC01269=-7.6002,0.0000
EC01270=-4.6784,0.0000
EC01271=-2.0841,0.0000
EC01272=0.0000,0.0000
EC01273=0.0000,0.0000
EC01274=2.0177,0.0000
EC01275=4.5896,0.0000
EC01276=7.5288,0.0000
EC01277=8.4644,0.0000
EC01278=8.5281,0.0000
EC01279=8.4283,0.0000
EC01280=8.3383,0.0000
EC01281=8.4379,0.0000
EC01282=10.0717,0.0000
EC01283=12.9390,0.0000
EC01284=16.5485,0.0000
EC01285=20.4866,0.0000
EC01286=24.5131,0.0000
EC01287=28.4517,0.0000
EC01288=32.0609,0.0000
EC01289=34.9281,0.0000
EC01290=36.5622,0.0000
EC01291=36.6621,0.0000
EC01292=36.5714,0.0000
EC01293=36.4714,0.0000
EC01294=36.5356,0.0000
EC01295=37.4711,0.0000
EC01296=40.4108,0.0000
EC01297=42.9827,0.0000
EC01298=45.0000,0.0000
EC01299=47.0166,0.0000
EC01300=49.5906,0.0000
EC01301=52.5289,0.0000
EC01302=53.4644,0.0000
EC01303=53.5286,0.0000
EC01304=53.4286,0.0000
EC01305=53.3379,0.0000
EC01306=53.4378,0.0000
EC01307=55.0719,0.0000
EC01308=57.9391,0.0000
EC01309=61.5483,0.0000
EC01310=65.4869,0.0000
EC01311=69.5134,0.0000
EC01312=73.4515,0.0000
EC01313=77.0610,0.0000
EC01314=79.9283,0.0000
EC01315=81.5621,0.0000
EC01316=81.6617,0.0000
EC01317=81.5717,0.0000
EC01318=81.4719,0.0000
EC01319=81.5356,0.0000
EC01320=82.4712,0.0000
EC01321=85.4104,0.0000
EC01322=87.9823,0.0000
EC01323=90.0000,0.0000
EC01324=92.0167,0.0000
EC01325=94.5896,0.0000
EC01326=97.5286,0.0000
EC01327=98.4644,0.0000
EC01328=98.5281,0.0000
EC01329=98.4283,0.0000
EC01330=98.3383,0.0000
EC01331=98.4379,0.0000
EC01332=100.0717,0.0000
EC01333=102.9390,0.0000
EC01334=106.5485,0.0000
EC01335=110.4866,0.0000
EC01336=114.5131,0.0000
EC01337=118.4517,0.0000
EC01338=122.0609,0.0000
EC01339=124.9281,0.0000
EC01340=126.5622,0.0000
EC01341=126.6621,0.0000
EC01342=126.5714,0.0000
EC01343=126.4714,0.0000
EC01344=126.5356,0.0000
EC01345=127.4711,0.0000
EC01346=130.4108,0.0000
EC01347=132.9827,0.0000
EC01348=135.0000,0.0000
EC01349=137.0166,0.0000
EC01350=139.5906,0.0000
EC01351=142.5289,0.0000
EC01352=143.4644,0.0000
EC01353=143.5286,0.0000
EC01354=143.4286,0.0000
EC01355=143.3379,0.0000
EC01356=143.4378,0.0000
EC01357=145.0719,0.0000
EC01358=147.9391,0.0000
EC01359=151.5483,0.0000
EC01360=155.4869,0.0000
EC01361=159.5134,0.0000
EC01362=163.4515,0.0000
EC01363=167.0610,0.0000
EC01364=169.9283,0.0000
EC01365=171.5621,0.0000
EC01366=171.6617,0.0000
EC01367=171.5717,0.0000
EC01368=171.4719,0.0000
EC01369=171.5356,0.0000
EC01370=172.4712,0.0000
EC01371=175.4104,0.0000
EC01372=177.9823,0.0000
EC01373=180.0000,0.0000
EC01374=180.0000,0.0000
EC01375=-177.9833,0.0000
EC01376=-175.4104,0.0000
EC01377=-172.4714,0.0000
EC01378=-171.5356,0.0000
EC01379=-171.4719,0.0000
EC01380=-171.5717,0.0000
EC01381=-171.6617,0.0000
EC01382=-171.5621,0.0000
EC01383=-169.9283,0.0000
EC01384=-167.0610,0.0000
EC01385=-163.4515,0.0000
EC01386=-159.5134,0.0000
EC01387=-155.4869,0.0000
EC01388=-151.5483,0.0000
EC01389=-147.9391,0.0000
EC01390=-145.0719,0.0000
EC01391=-143.4378,0.0000
EC01392=-143.3379,0.0000
EC01393=-143.4286,0.0000
EC01394=-143.5286,0.0000
EC01395=-143.4644,0.0000
EC01396=-142.5289,0.0000
EC01397=-139.5892,0.0000
EC01398=-137.0173,0.0000
EC01399=-135.0000,0.0000
EC01400=-132.9834,0.0000
EC01401=-130.4094,0.0000
EC01402=-127.4711,0.0000
EC01403=-126.5356,0.0000
EC01404=-126.4714,0.0000
EC01405=-126.5714,0.0000
EC01406=-126.6621,0.0000
EC01407=-126.5622,0.0000
EC01408=-124.9281,0.0000
EC01409=-122.0609,0.0000
EC01410=-118.4517,0.0000
EC01411=-114.5131,0.0000
EC01412=-110.4866,0.0000
EC01413=-106.5485,0.0000
EC01414=-102.9390,0.0000
EC01415=-100.0717,0.0000
EC01416=-98.4379,0.0000
EC01417=-98.3383,0.0000
EC01418=-98.4283,0.0000
EC01419=-98.5281,0.0000
EC01420=-98.4644,0.0000
EC01421=-97.5288,0.0000
EC01422=-94.5896,0.0000
EC01423=-92.0177,0.0000
EC01424=-90.0000,0.0000
EC01425=-87.9833,0.0000
EC01426=-85.4104,0.0000
EC01427=-82.4714,0.0000
EC01428=-81.5356,0.0000
EC01429=-81.4719,0.0000
EC01430=-81.5717,0.0000
EC01431=-81.6617,0.0000
EC01432=-81.5621,0.0000
EC01433=-79.9283,0.0000
EC01434=-77.0610,0.0000
EC01435=-73.4515,0.0000
EC01436=-69.5134,0.0000
EC01437=-65.4869,0.0000
EC01438=-61.5483,0.0000
EC01439=-57.9391,0.0000
EC01440=-55.0719,0.0000
EC01441=-53.4378,0.0000
EC01442=-53.3379,0.0000
EC01443=-53.4286,0.0000
EC01444=-53.5286,0.0000
EC01445=-53.4644,0.0000
EC01446=-52.5289,0.0000
EC01447=-49.5892,0.0000
EC01448=-47.0173,0.0000
EC01449=-45.0000,0.0000
EC01450=-42.9834,0.0000
EC01451=-40.4094,0.0000
EC01452=-37.4711,0.0000
EC01453=-36.5356,0.0000
EC01454=-36.4714,0.0000
EC01455=-36.5714,0.0000
EC01456=-36.6621,0.0000
EC01457=-36.5622,0.0000
EC01458=-34.9281,0.0000
EC01459=-32.0609,0.0000
EC01460=-28.4517,0.0000
EC01461=-24.5131,0.0000
EC01462=-20.4866,0.0000
EC01463=-16.5485,0.0000
EC01464=-12.9390,0.0000
EC01465=-10.0717,0.0000
EC01466=-8.4379,0.0000
EC01467=-8.3383,0.0000
EC01468=-8.4283,0.0000
EC01469=-8.5281,0.0000
EC01470=-8.4644,0.0000
EC01471=-7.5286,0.0000
EC01472=-4.5896,0.0000
EC01473=-2.0167,0.0000
EC01474=0.0000,0.0000
EC01475=0.0000,0.0000
EC01476=1.9494,0.0000
EC01477=4.4996,0.0000
EC01478=7.4570,0.0000
EC01479=8.3570,0.0000
EC01480=8.3879,0.0000
EC01481=8.2735,0.0000
EC01482=8.1767,0.0000
EC01483=8.2659,0.0000
EC01484=9.9145,0.0000
EC01485=12.8156,0.0000
EC01486=16.4700,0.0000
EC01487=20.4601,0.0000
EC01488=24.5401,0.0000
EC01489=28.5303,0.0000
EC01490=32.1847,0.0000
EC01491=35.0854,0.0000
EC01492=36.7338,0.0000
EC01493=36.8229,0.0000
EC01494=36.7263,0.0000
EC01495=36.6122,0.0000
EC01496=36.6435,0.0000
EC01497=37.5429,0.0000
EC01498=40.5003,0.0000
EC01499=43.0512,0.0000
EC01500=45.0000,0.0000
EC01501=46.9488,0.0000
EC01502=49.5003,0.0000
EC01503=52.4571,0.0000
EC01504=53.3565,0.0000
EC01505=53.3878,0.0000
EC01506=53.2737,0.0000
EC01507=53.1771,0.0000
EC01508=53.2662,0.0000
EC01509=54.9146,0.0000
EC01510=57.8153,0.0000
EC01511=61.4697,0.0000
EC01512=65.4599,0.0000
EC01513=69.5399,0.0000
EC01514=73.5300,0.0000
EC01515=77.1844,0.0000
EC01516=80.0855,0.0000
EC01517=81.7341,0.0000
EC01518=81.8233,0.0000
EC01519=81.7265,0.0000
EC01520=81.6121,0.0000
EC01521=81.6430,0.0000
EC01522=82.5430,0.0000
EC01523=85.5004,0.0000
EC01524=88.0506,0.0000
EC01525=90.0000,0.0000
EC01526=91.9484,0.0000
EC01527=94.5006,0.0000
EC01528=97.4570,0.0000
EC01529=98.3570,0.0000
EC01530=98.3879,0.0000
EC01531=98.2735,0.0000
EC01532=98.1767,0.0000
EC01533=98.2659,0.0000
EC01534=99.9145,0.0000
EC01535=102.8156,0.0000
EC01536=106.4700,0.0000
EC01537=110.4601,0.0000
EC01538=114.5401,0.0000
EC01539=118.5303,0.0000
EC01540=122.1847,0.0000
EC01541=125.0854,0.0000
EC01542=126.7338,0.0000
EC01543=126.8229,0.0000
EC01544=126.7263,0.0000
EC01545=126.6122,0.0000
EC01546=126.6435,0.0000
EC01547=127.5429,0.0000
EC01548=130.5003,0.0000
EC01549=133.0512,0.0000
EC01550=135.0000,0.0000
EC01551=136.9488,0.0000
EC01552=139.5003,0.0000
EC01553=142.4571,0.0000
EC01554=143.3565,0.0000
EC01555=143.3878,0.0000
EC01556=143.2737,0.0000
EC01557=143.1771,0.0000
EC01558=143.2662,0.0000
EC01559=144.9146,0.0000
EC01560=147.8153,0.0000
EC01561=151.4697,0.0000
EC01562=155.4599,0.0000
EC01563=159.5399,0.0000
EC01564=163.5300,0.0000
EC01565=167.1844,0.0000
EC01566=170.0855,0.0000
EC01567=171.7341,0.0000
EC01568=171.8233,0.0000
EC01569=171.7265,0.0000
EC01570=171.6121,0.0000
EC01571=171.6430,0.0000
EC01572=172.5430,0.0000
EC01573=175.5004,0.0000
EC01574=178.0506,0.0000
EC01575=180.0000,0.0000
EC01576=180.0000,0.0000
EC01577=-178.0516,0.0000
EC01578=-175.4994,0.0000
EC01579=-172.5430,0.0000
EC01580=-171.6430,0.0000
EC01581=-171.6121,0.0000
EC01582=-171.7265,0.0000
EC01583=-171.8233,0.0000
EC01584=-171.7341,0.0000
EC01585=-170.0855,0.0000
EC01586=-167.1844,0.0000
EC01587=-163.5300,0.0000
EC01588=-159.5399,0.0000
EC01589=-155.4599,0.0000
EC01590=-151.4697,0.0000
EC01591=-147.8153,0.0000
EC01592=-144.9146,0.0000
EC01593=-143.2662,0.0000
EC01594=-143.1771,0.0000
EC01595=-143.2737,0.0000
EC01596=-143.3878,0.0000
EC01597=-143.3565,0.0000
EC01598=-142.4571,0.0000
EC01599=-139.4997,0.0000
EC01600=-136.9488,0.0000
EC01601=-135.0000,0.0000
EC01602=-133.0512,0.0000
EC01603=-130.4997,0.0000
EC01604=-127.5429,0.0000
EC01605=-126.6435,0.0000
EC01606=-126.6122,0.0000
EC01607=-126.7263,0.0000
EC01608=-126.8229,0.0000
EC01609=-126.7338,0.0000
EC01610=-125.0854,0.0000
EC01611=-122.1847,0.0000
EC01612=-118.5303,0.0000
EC01613=-114.5401,0.0000
EC01614=-110.4601,0.0000
EC01615=-106.4700,0.0000
EC01616=-102.8156,0.0000
EC01617=-99.9145,0.0000
EC01618=-98.2659,0.0000
EC01619=-98.1767,0.0000
EC01620=-98.2735,0.0000
EC01621=-98.3879,0.0000
EC01622=-98.3570,0.0000
EC01623=-97.4570,0.0000
EC01624=-94.4996,0.0000
EC01625=-91.9494,0.0000
EC01626=-90.0000,0.0000
EC01627=-88.0516,0.0000
EC01628=-85.4994,0.0000
EC01629=-82.5430,0.0000
EC01630=-81.6430,0.0000
EC01631=-81.6121,0.0000
EC01632=-81.7265,0.0000
EC01633=-81.8233,0.0000
EC01634=-81.7341,0.0000
EC01635=-80.0855,0.0000
EC01636=-77.1844,0.0000
EC01637=-73.5300,0.0000
EC01638=-69.5399,0.0000
EC01639=-65.4599,0.0000
EC01640=-61.4697,0.0000
EC01641=-57.8153,0.0000
EC01642=-54.9146,0.0000
EC01643=-53.2662,0.0000
EC01644=-53.1771,0.0000
EC01645=-53.2737,0.0000
EC01646=-53.3878,0.0000
EC01647=-53.3565,0.0000
EC01648=-52.4571,0.0000
EC01649=-49.4997,0.0000
EC01650=-46.9488,0.0000
EC01651=-45.0000,0.0000
EC01652=-43.0512,0.0000
EC01653=-40.4997,0.0000
EC01654=-37.5429,0.0000
EC01655=-36.6435,0.0000
EC01656=-36.6122,0.0000
EC01657=-36.7263,0.0000
EC01658=-36.8229,0.0000
EC01659=-36.7338,0.0000
EC01660=-35.0854,0.0000
EC01661=-32.1847,0.0000
EC01662=-28.5303,0.0000
EC01663=-24.5401,0.0000
EC01664=-20.4601,0.0000
EC01665=-16.4700,0.0000
EC01666=-12.8156,0.0000
EC01667=-9.9145,0.0000
EC01668=-8.2659,0.0000
EC01669=-8.1767,0.0000
EC01670=-8.2735,0.0000
EC01671=-8.3879,0.0000
EC01672=-8.3570,0.0000
EC01673=-7.4570,0.0000
EC01674=-4.5006,0.0000
EC01675=-1.9484,0.0000
EC01676=0.0000,0.0000
EC01677=0.0000,0.0000
EC01678=1.8799,0.0000
EC01679=4.4091,0.0000
EC01680=7.3837,0.0000
EC01681=8.2508,0.0000
EC01682=8.2514,0.0000
EC01683=8.1286,0.0000
EC01684=8.0287,0.0000
EC01685=8.1105,0.0000
EC01686=9.7738,0.0000
EC01687=12.7052,0.0000
EC01688=16.4001,0.0000
EC01689=20.4362,0.0000
EC01690=24.5637,0.0000
EC01691=28.5997,0.0000
EC01692=32.2952,0.0000
EC01693=35.2262,0.0000
EC01694=36.8889,0.0000
EC01695=36.9711,0.0000
EC01696=36.8716,0.0000
EC01697=36.7487,0.0000
EC01698=36.7500,0.0000
EC01699=37.6160,0.0000
EC01700=40.5914,0.0000
EC01701=43.1202,0.0000
EC01702=45.0000,0.0000
EC01703=46.8791,0.0000
EC01704=49.4092,0.0000
EC01705=52.3840,0.0000
EC01706=53.2500,0.0000
EC01707=53.2513,0.0000
EC01708=53.1284,0.0000
EC01709=53.0289,0.0000
EC01710=53.1111,0.0000
EC01711=54.7738,0.0000
EC01712=57.7048,0.0000
EC01713=61.4003,0.0000
EC01714=65.4363,0.0000
EC01715=69.5638,0.0000
EC01716=73.5999,0.0000
EC01717=77.2948,0.0000
EC01718=80.2262,0.0000
EC01719=81.8895,0.0000
EC01720=81.9713,0.0000
EC01721=81.8714,0.0000
EC01722=81.7486,0.0000
EC01723=81.7492,0.0000
EC01724=82.6163,0.0000
EC01725=85.5909,0.0000
EC01726=88.1201,0.0000
EC01727=90.0000,0.0000
EC01728=91.8799,0.0000
EC01729=94.4091,0.0000
EC01730=97.3837,0.0000
EC01731=98.2508,0.0000
EC01732=98.2514,0.0000
EC01733=98.1286,0.0000
EC01734=98.0287,0.0000
EC01735=98.1105,0.0000
EC01736=99.7738,0.0000
EC01737=102.7052,0.0000
EC01738=106.4001,0.0000
EC01739=110.4362,0.0000
EC01740=114.5637,0.0000
EC01741=118.5997,0.0000
EC01742=122.2952,0.0000
EC01743=125.2262,0.0000
EC01744=126.8889,0.0000
EC01745=126.9711,0.0000
EC01746=126.8716,0.0000
EC01747=126.7487,0.0000
EC01748=126.7500,0.0000
EC01749=127.6160,0.0000
EC01750=130.5914,0.0000
EC01751=133.1202,0.0000
EC01752=135.0000,0.0000
EC01753=136.8791,0.0000
EC01754=139.4092,0.0000
EC01755=142.3840,0.0000
EC01756=143.2500,0.0000
EC01757=143.2513,0.0000
EC01758=143.1284,0.0000
EC01759=143.0289,0.0000
EC01760=143.1111,0.0000
EC01761=144.7738,0.0000
EC01762=147.7048,0.0000
EC01763=151.4003,0.0000
EC01764=155.4363,0.0000
EC01765=159.5638,0.0000
EC01766=163.5999,0.0000
EC01767=167.2948,0.0000
EC01768=170.2262,0.0000
EC01769=171.8895,0.0000
EC01770=171.9713,0.0000
EC01771=171.8714,0.0000
EC01772=171.7486,0.0000
EC01773=171.7492,0.0000
EC01774=172.6163,0.0000
EC01775=175.5909,0.0000
EC01776=178.1201,0.0000
EC01777=180.0000,0.0000
EC01778=180.0000,0.0000
EC01779=-178.1201,0.0000
EC01780=-175.5909,0.0000
EC01781=-172.6163,0.0000
EC01782=-171.7492,0.0000
EC01783=-171.7486,0.0000
EC01784=-171.8714,0.0000
EC01785=-171.9713,0.0000
EC01786=-171.8895,0.0000
EC01787=-170.2262,0.0000
EC01788=-167.2948,0.0000
EC01789=-163.5999,0.0000
EC01790=-159.5638,0.0000
EC01791=-155.4363,0.0000
EC01792=-151.4003,0.0000
EC01793=-147.7048,0.0000
EC01794=-144.7738,0.0000
EC01795=-143.1111,0.0000
EC01796=-143.0289,0.0000
EC01797=-143.1284,0.0000
EC01798=-143.2513,0.0000
EC01799=-143.2500,0.0000
EC01800=-142.3840,0.0000
EC01801=-139.4086,0.0000
EC01802=-136.8798,0.0000
EC01803=-135.0000,0.0000
EC01804=-133.1209,0.0000
EC01805=-130.5908,0.0000
EC01806=-127.6160,0.0000
EC01807=-126.7500,0.0000
EC01808=-126.7487,0.0000
EC01809=-126.8716,0.0000
EC01810=-126.9711,0.0000
EC01811=-126.8889,0.0000
EC01812=-125.2262,0.0000
EC01813=-122.2952,0.0000
EC01814=-118.5997,0.0000
EC01815=-114.5637,0.0000
EC01816=-110.4362,0.0000
EC01817=-106.4001,0.0000
EC01818=-102.7052,0.0000
EC01819=-99.7738,0.0000
EC01820=-98.1105,0.0000
EC01821=-98.0287,0.0000
EC01822=-98.1286,0.0000
EC01823=-98.2514,0.0000
EC01824=-98.2508,0.0000
EC01825=-97.3837,0.0000
EC01826=-94.4091,0.0000
EC01827=-91.8799,0.0000
EC01828=-90.0000,0.0000
EC01829=-88.1201,0.0000
EC01830=-85.5909,0.0000
EC01831=-82.6163,0.0000
EC01832=-81.7492,0.0000
EC01833=-81.7486,0.0000
EC01834=-81.8714,0.0000
EC01835=-81.9713,0.0000
EC01836=-81.8895,0.0000
EC01837=-80.2262,0.0000
EC01838=-77.2948,0.0000
EC01839=-73.5999,0.0000
EC01840=-69.5638,0.0000
EC01841=-65.4363,0.0000
EC01842=-61.4003,0.0000
EC01843=-57.7048,0.0000
EC01844=-54.7738,0.0000
EC01845=-53.1111,0.0000
EC01846=-53.0289,0.0000
EC01847=-53.1284,0.0000
EC01848=-53.2513,0.0000
EC01849=-53.2500,0.0000
EC01850=-52.3840,0.0000
EC01851=-49.4086,0.0000
EC01852=-46.8798,0.0000
EC01853=-45.0000,0.0000
EC01854=-43.1209,0.0000
EC01855=-40.5908,0.0000
EC01856=-37.6160,0.0000
EC01857=-36.7500,0.0000
EC01858=-36.7487,0.0000
EC01859=-36.8716,0.0000
EC01860=-36.9711,0.0000
EC01861=-36.8889,0.0000
EC01862=-35.2262,0.0000
EC01863=-32.2952,0.0000
EC01864=-28.5997,0.0000
EC01865=-24.5637,0.0000
EC01866=-20.4362,0.0000
EC01867=-16.4001,0.0000
EC01868=-12.7052,0.0000
EC01869=-9.7738,0.0000
EC01870=-8.1105,0.0000
EC01871=-8.0287,0.0000
EC01872=-8.1286,0.0000
EC01873=-8.2514,0.0000
EC01874=-8.2508,0.0000
EC01875=-7.3837,0.0000
EC01876=-4.4091,0.0000
EC01877=-1.8799,0.0000
EC01878=0.0000,0.0000
EC01879=0.0000,0.0000
EC01880=1.8104,0.0000
EC01881=4.3168,0.0000
EC01882=7.3110,0.0000
EC01883=8.1459,0.0000
EC01884=8.1209,0.0000
EC01885=7.9932,0.0000
EC01886=7.8955,0.0000
EC01887=7.9733,0.0000
EC01888=9.6504,0.0000
EC01889=12.6088,0.0000
EC01890=16.3398,0.0000
EC01891=20.4161,0.0000
EC01892=24.5839,0.0000
EC01893=28.6599,0.0000
EC01894=32.3913,0.0000
EC01895=35.3500,0.0000
EC01896=37.0265,0.0000
EC01897=37.1043,0.0000
EC01898=37.0066,0.0000
EC01899=36.8795,0.0000
EC01900=36.8537,0.0000
EC01901=37.6887,0.0000
EC01902=40.6829,0.0000
EC01903=43.1899,0.0000
EC01904=45.0000,0.0000
EC01905=46.8101,0.0000
EC01906=49.3178,0.0000
EC01907=52.3119,0.0000
EC01908=53.1463,0.0000
EC01909=53.1205,0.0000
EC01910=52.9934,0.0000
EC01911=52.8957,0.0000
EC01912=52.9735,0.0000
EC01913=54.6500,0.0000
EC01914=57.6087,0.0000
EC01915=61.3401,0.0000
EC01916=65.4161,0.0000
EC01917=69.5839,0.0000
EC01918=73.6602,0.0000
EC01919=77.3912,0.0000
EC01920=80.3496,0.0000
EC01921=82.0267,0.0000
EC01922=82.1045,0.0000
EC01923=82.0068,0.0000
EC01924=81.8791,0.0000
EC01925=81.8541,0.0000
EC01926=82.6890,0.0000
EC01927=85.6832,0.0000
EC01928=88.1896,0.0000
EC01929=90.0000,0.0000
EC01930=91.8094,0.0000
EC01931=94.3178,0.0000
EC01932=97.3110,0.0000
EC01933=98.1459,0.0000
EC01934=98.1209,0.0000
EC01935=97.9932,0.0000
EC01936=97.8955,0.0000
EC01937=97.9733,0.0000
EC01938=99.6504,0.0000
EC01939=102.6088,0.0000
EC01940=106.3398,0.0000
EC01941=110.4161,0.0000
EC01942=114.5839,0.0000
EC01943=118.6599,0.0000
EC01944=122.3913,0.0000
EC01945=125.3500,0.0000
EC01946=127.0265,0.0000
EC01947=127.1043,0.0000
EC01948=127.0066,0.0000
EC01949=126.8795,0.0000
EC01950=126.8537,0.0000
EC01951=127.6887,0.0000
EC01952=130.6829,0.0000
EC01953=133.1899,0.0000
EC01954=135.0000,0.0000
EC01955=136.8101,0.0000
EC01956=139.3178,0.0000
EC01957=142.3119,0.0000
EC01958=143.1463,0.0000
EC01959=143.1205,0.0000
EC01960=142.9934,0.0000
EC01961=142.8957,0.0000
EC01962=142.9735,0.0000
EC01963=144.6500,0.0000
EC01964=147.6087,0.0000
EC01965=151.3401,0.0000
EC01966=155.4161,0.0000
EC01967=159.5839,0.0000
EC01968=163.6602,0.0000
EC01969=167.3912,0.0000
EC01970=170.3496,0.0000
EC01971=172.0267,0.0000
EC01972=172.1045,0.0000
EC01973=172.0068,0.0000
EC01974=171.8791,0.0000
EC01975=171.8541,0.0000
EC01976=172.6890,0.0000
EC01977=175.6832,0.0000
EC01978=178.1896,0.0000
EC01979=180.0000,0.0000
EC01980=180.0000,0.0000
EC01981=-178.1906,0.0000
EC01982=-175.6822,0.0000
EC01983=-172.6890,0.0000
EC01984=-171.8541,0.0000
EC01985=-171.8791,0.0000
EC01986=-172.0068,0.0000
EC01987=-172.1045,0.0000
EC01988=-172.0267,0.0000
EC01989=-170.3496,0.0000
EC01990=-167.3912,0.0000
EC01991=-163.6602,0.0000
EC01992=-159.5839,0.0000
EC01993=-155.4161,0.0000
EC01994=-151.3401,0.0000
EC01995=-147.6087,0.0000
EC01996=-144.6500,0.0000
EC01997=-142.9735,0.0000
EC01998=-142.8957,0.0000
EC01999=-142.9934,0.0000
//INST
///DATE 2021/02/10 13:51
///COMM
///ATTR SC,RW,RJ
////FRAME USER 2
///GROUP1 RB1
///GROUP2 ST1
NOP
SMOVL C00000 +MOVJ EC00000
SMOVL C00001 +MOVJ EC00001
SMOVL C00002 +MOVJ EC00002
SMOVL C00003 +MOVJ EC00003
SMOVL C00004 +MOVJ EC00004
SMOVL C00005 +MOVJ EC00005
SMOVL C00006 +MOVJ EC00006
SMOVL C00007 +MOVJ EC00007
SMOVL C00008 +MOVJ EC00008
SMOVL C00009 +MOVJ EC00009
SMOVL C00010 +MOVJ EC00010
SMOVL C00011 +MOVJ EC00011
SMOVL C00012 +MOVJ EC00012
SMOVL C00013 +MOVJ EC00013
SMOVL C00014 +MOVJ EC00014
SMOVL C00015 +MOVJ EC00015
SMOVL C00016 +MOVJ EC00016
SMOVL C00017 +MOVJ EC00017
SMOVL C00018 +MOVJ EC00018
SMOVL C00019 +MOVJ EC00019
SMOVL C00020 +MOVJ EC00020
SMOVL C00021 +MOVJ EC00021
SMOVL C00022 +MOVJ EC00022
SMOVL C00023 +MOVJ EC00023
SMOVL C00024 +MOVJ EC00024
SMOVL C00025 +MOVJ EC00025
SMOVL C00026 +MOVJ EC00026
SMOVL C00027 +MOVJ EC00027
SMOVL C00028 +MOVJ EC00028
SMOVL C00029 +MOVJ EC00029
SMOVL C00030 +MOVJ EC00030
SMOVL C00031 +MOVJ EC00031
SMOVL C00032 +MOVJ EC00032
SMOVL C00033 +MOVJ EC00033
SMOVL C00034 +MOVJ EC00034
SMOVL C00035 +MOVJ EC00035
SMOVL C00036 +MOVJ EC00036
SMOVL C00037 +MOVJ EC00037
SMOVL C00038 +MOVJ EC00038
SMOVL C00039 +MOVJ EC00039
SMOVL C00040 +MOVJ EC00040
SMOVL C00041 +MOVJ EC00041
SMOVL C00042 +MOVJ EC00042
SMOVL C00043 +MOVJ EC00043
SMOVL C00044 +MOVJ EC00044
SMOVL C00045 +MOVJ EC00045
SMOVL C00046 +MOVJ EC00046
SMOVL C00047 +MOVJ EC00047
SMOVL C00048 +MOVJ EC00048
SMOVL C00049 +MOVJ EC00049
SMOVL C00050 +MOVJ EC00050
SMOVL C00051 +MOVJ EC00051
SMOVL C00052 +MOVJ EC00052
SMOVL C00053 +MOVJ EC00053
SMOVL C00054 +MOVJ EC00054
SMOVL C00055 +MOVJ EC00055
SMOVL C00056 +MOVJ EC00056
SMOVL C00057 +MOVJ EC00057
SMOVL C00058 +MOVJ EC00058
SMOVL C00059 +MOVJ EC00059
SMOVL C00060 +MOVJ EC00060
SMOVL C00061 +MOVJ EC00061
SMOVL C00062 +MOVJ EC00062
SMOVL C00063 +MOVJ EC00063
SMOVL C00064 +MOVJ EC00064
SMOVL C00065 +MOVJ EC00065
SMOVL C00066 +MOVJ EC00066
SMOVL C00067 +MOVJ EC00067
SMOVL C00068 +MOVJ EC00068
SMOVL C00069 +MOVJ EC00069
SMOVL C00070 +MOVJ EC00070
SMOVL C00071 +MOVJ EC00071
SMOVL C00072 +MOVJ EC00072
SMOVL C00073 +MOVJ EC00073
SMOVL C00074 +MOVJ EC00074
SMOVL C00075 +MOVJ EC00075
SMOVL C00076 +MOVJ EC00076
SMOVL C00077 +MOVJ EC00077
SMOVL C00078 +MOVJ EC00078
SMOVL C00079 +MOVJ EC00079
SMOVL C00080 +MOVJ EC00080
SMOVL C00081 +MOVJ EC00081
SMOVL C00082 +MOVJ EC00082
SMOVL C00083 +MOVJ EC00083
SMOVL C00084 +MOVJ EC00084
SMOVL C00085 +MOVJ EC00085
SMOVL C00086 +MOVJ EC00086
SMOVL C00087 +MOVJ EC00087
SMOVL C00088 +MOVJ EC00088
SMOVL C00089 +MOVJ EC00089
SMOVL C00090 +MOVJ EC00090
SMOVL C00091 +MOVJ EC00091
SMOVL C00092 +MOVJ EC00092
SMOVL C00093 +MOVJ EC00093
SMOVL C00094 +MOVJ EC00094
SMOVL C00095 +MOVJ EC00095
SMOVL C00096 +MOVJ EC00096
SMOVL C00097 +MOVJ EC00097
SMOVL C00098 +MOVJ EC00098
SMOVL C00099 +MOVJ EC00099
SMOVL C00100 +MOVJ EC00100
SMOVL C00101 +MOVJ EC00101
SMOVL C00102 +MOVJ EC00102
SMOVL C00103 +MOVJ EC00103
SMOVL C00104 +MOVJ EC00104
SMOVL C00105 +MOVJ EC00105
SMOVL C00106 +MOVJ EC00106
SMOVL C00107 +MOVJ EC00107
SMOVL C00108 +MOVJ EC00108
SMOVL C00109 +MOVJ EC00109
SMOVL C00110 +MOVJ EC00110
SMOVL C00111 +MOVJ EC00111
SMOVL C00112 +MOVJ EC00112
SMOVL C00113 +MOVJ EC00113
SMOVL C00114 +MOVJ EC00114
SMOVL C00115 +MOVJ EC00115
SMOVL C00116 +MOVJ EC00116
SMOVL C00117 +MOVJ EC00117
SMOVL C00118 +MOVJ EC00118
SMOVL C00119 +MOVJ EC00119
SMOVL C00120 +MOVJ EC00120
SMOVL C00121 +MOVJ EC00121
SMOVL C00122 +MOVJ EC00122
SMOVL C00123 +MOVJ EC00123
SMOVL C00124 +MOVJ EC00124
SMOVL C00125 +MOVJ EC00125
SMOVL C00126 +MOVJ EC00126
SMOVL C00127 +MOVJ EC00127
SMOVL C00128 +MOVJ EC00128
SMOVL C00129 +MOVJ EC00129
SMOVL C00130 +MOVJ EC00130
SMOVL C00131 +MOVJ EC00131
SMOVL C00132 +MOVJ EC00132
SMOVL C00133 +MOVJ EC00133
SMOVL C00134 +MOVJ EC00134
SMOVL C00135 +MOVJ EC00135
SMOVL C00136 +MOVJ EC00136
SMOVL C00137 +MOVJ EC00137
SMOVL C00138 +MOVJ EC00138
SMOVL C00139 +MOVJ EC00139
SMOVL C00140 +MOVJ EC00140
SMOVL C00141 +MOVJ EC00141
SMOVL C00142 +MOVJ EC00142
SMOVL C00143 +MOVJ EC00143
SMOVL C00144 +MOVJ EC00144
SMOVL C00145 +MOVJ EC00145
SMOVL C00146 +MOVJ EC00146
SMOVL C00147 +MOVJ EC00147
SMOVL C00148 +MOVJ EC00148
SMOVL C00149 +MOVJ EC00149
SMOVL C00150 +MOVJ EC00150
SMOVL C00151 +MOVJ EC00151
SMOVL C00152 +MOVJ EC00152
SMOVL C00153 +MOVJ EC00153
SMOVL C00154 +MOVJ EC00154
SMOVL C00155 +MOVJ EC00155
SMOVL C00156 +MOVJ EC00156
SMOVL C00157 +MOVJ EC00157
SMOVL C00158 +MOVJ EC00158
SMOVL C00159 +MOVJ EC00159
SMOVL C00160 +MOVJ EC00160
SMOVL C00161 +MOVJ EC00161
SMOVL C00162 +MOVJ EC00162
SMOVL C00163 +MOVJ EC00163
SMOVL C00164 +MOVJ EC00164
SMOVL C00165 +MOVJ EC00165
SMOVL C00166 +MOVJ EC00166
SMOVL C00167 +MOVJ EC00167
SMOVL C00168 +MOVJ EC00168
SMOVL C00169 +MOVJ EC00169
SMOVL C00170 +MOVJ EC00170
SMOVL C00171 +MOVJ EC00171
SMOVL C00172 +MOVJ EC00172
SMOVL C00173 +MOVJ EC00173
SMOVL C00174 +MOVJ EC00174
SMOVL C00175 +MOVJ EC00175
SMOVL C00176 +MOVJ EC00176
SMOVL C00177 +MOVJ EC00177
SMOVL C00178 +MOVJ EC00178
SMOVL C00179 +MOVJ EC00179
SMOVL C00180 +MOVJ EC00180
SMOVL C00181 +MOVJ EC00181
SMOVL C00182 +MOVJ EC00182
SMOVL C00183 +MOVJ EC00183
SMOVL C00184 +MOVJ EC00184
SMOVL C00185 +MOVJ EC00185
SMOVL C00186 +MOVJ EC00186
SMOVL C00187 +MOVJ EC00187
SMOVL C00188 +MOVJ EC00188
SMOVL C00189 +MOVJ EC00189
SMOVL C00190 +MOVJ EC00190
SMOVL C00191 +MOVJ EC00191
SMOVL C00192 +MOVJ EC00192
SMOVL C00193 +MOVJ EC00193
SMOVL C00194 +MOVJ EC00194
SMOVL C00195 +MOVJ EC00195
SMOVL C00196 +MOVJ EC00196
SMOVL C00197 +MOVJ EC00197
SMOVL C00198 +MOVJ EC00198
SMOVL C00199 +MOVJ EC00199
SMOVL C00200 +MOVJ EC00200
SMOVL C00201 +MOVJ EC00201
SMOVL C00202 +MOVJ EC00202
SMOVL C00203 +MOVJ EC00203
SMOVL C00204 +MOVJ EC00204
SMOVL C00205 +MOVJ EC00205
SMOVL C00206 +MOVJ EC00206
SMOVL C00207 +MOVJ EC00207
SMOVL C00208 +MOVJ EC00208
SMOVL C00209 +MOVJ EC00209
SMOVL C00210 +MOVJ EC00210
SMOVL C00211 +MOVJ EC00211
SMOVL C00212 +MOVJ EC00212
SMOVL C00213 +MOVJ EC00213
SMOVL C00214 +MOVJ EC00214
SMOVL C00215 +MOVJ EC00215
SMOVL C00216 +MOVJ EC00216
SMOVL C00217 +MOVJ EC00217
SMOVL C00218 +MOVJ EC00218
SMOVL C00219 +MOVJ EC00219
SMOVL C00220 +MOVJ EC00220
SMOVL C00221 +MOVJ EC00221
SMOVL C00222 +MOVJ EC00222
SMOVL C00223 +MOVJ EC00223
SMOVL C00224 +MOVJ EC00224
SMOVL C00225 +MOVJ EC00225
SMOVL C00226 +MOVJ EC00226
SMOVL C00227 +MOVJ EC00227
SMOVL C00228 +MOVJ EC00228
SMOVL C00229 +MOVJ EC00229
SMOVL C00230 +MOVJ EC00230
SMOVL C00231 +MOVJ EC00231
SMOVL C00232 +MOVJ EC00232
SMOVL C00233 +MOVJ EC00233
SMOVL C00234 +MOVJ EC00234
SMOVL C00235 +MOVJ EC00235
SMOVL C00236 +MOVJ EC00236
SMOVL C00237 +MOVJ EC00237
SMOVL C00238 +MOVJ EC00238
SMOVL C00239 +MOVJ EC00239
SMOVL C00240 +MOVJ EC00240
SMOVL C00241 +MOVJ EC00241
SMOVL C00242 +MOVJ EC00242
SMOVL C00243 +MOVJ EC00243
SMOVL C00244 +MOVJ EC00244
SMOVL C00245 +MOVJ EC00245
SMOVL C00246 +MOVJ EC00246
SMOVL C00247 +MOVJ EC00247
SMOVL C00248 +MOVJ EC00248
SMOVL C00249 +MOVJ EC00249
SMOVL C00250 +MOVJ EC00250
SMOVL C00251 +MOVJ EC00251
SMOVL C00252 +MOVJ EC00252
SMOVL C00253 +MOVJ EC00253
SMOVL C00254 +MOVJ EC00254
SMOVL C00255 +MOVJ EC00255
SMOVL C00256 +MOVJ EC00256
SMOVL C00257 +MOVJ EC00257
SMOVL C00258 +MOVJ EC00258
SMOVL C00259 +MOVJ EC00259
SMOVL C00260 +MOVJ EC00260
SMOVL C00261 +MOVJ EC00261
SMOVL C00262 +MOVJ EC00262
SMOVL C00263 +MOVJ EC00263
SMOVL C00264 +MOVJ EC00264
SMOVL C00265 +MOVJ EC00265
SMOVL C00266 +MOVJ EC00266
SMOVL C00267 +MOVJ EC00267
SMOVL C00268 +MOVJ EC00268
SMOVL C00269 +MOVJ EC00269
SMOVL C00270 +MOVJ EC00270
SMOVL C00271 +MOVJ EC00271
SMOVL C00272 +MOVJ EC00272
SMOVL C00273 +MOVJ EC00273
SMOVL C00274 +MOVJ EC00274
SMOVL C00275 +MOVJ EC00275
SMOVL C00276 +MOVJ EC00276
SMOVL C00277 +MOVJ EC00277
SMOVL C00278 +MOVJ EC00278
SMOVL C00279 +MOVJ EC00279
SMOVL C00280 +MOVJ EC00280
SMOVL C00281 +MOVJ EC00281
SMOVL C00282 +MOVJ EC00282
SMOVL C00283 +MOVJ EC00283
SMOVL C00284 +MOVJ EC00284
SMOVL C00285 +MOVJ EC00285
SMOVL C00286 +MOVJ EC00286
SMOVL C00287 +MOVJ EC00287
SMOVL C00288 +MOVJ EC00288
SMOVL C00289 +MOVJ EC00289
SMOVL C00290 +MOVJ EC00290
SMOVL C00291 +MOVJ EC00291
SMOVL C00292 +MOVJ EC00292
SMOVL C00293 +MOVJ EC00293
SMOVL C00294 +MOVJ EC00294
SMOVL C00295 +MOVJ EC00295
SMOVL C00296 +MOVJ EC00296
SMOVL C00297 +MOVJ EC00297
SMOVL C00298 +MOVJ EC00298
SMOVL C00299 +MOVJ EC00299
SMOVL C00300 +MOVJ EC00300
SMOVL C00301 +MOVJ EC00301
SMOVL C00302 +MOVJ EC00302
SMOVL C00303 +MOVJ EC00303
SMOVL C00304 +MOVJ EC00304
SMOVL C00305 +MOVJ EC00305
SMOVL C00306 +MOVJ EC00306
SMOVL C00307 +MOVJ EC00307
SMOVL C00308 +MOVJ EC00308
SMOVL C00309 +MOVJ EC00309
SMOVL C00310 +MOVJ EC00310
SMOVL C00311 +MOVJ EC00311
SMOVL C00312 +MOVJ EC00312
SMOVL C00313 +MOVJ EC00313
SMOVL C00314 +MOVJ EC00314
SMOVL C00315 +MOVJ EC00315
SMOVL C00316 +MOVJ EC00316
SMOVL C00317 +MOVJ EC00317
SMOVL C00318 +MOVJ EC00318
SMOVL C00319 +MOVJ EC00319
SMOVL C00320 +MOVJ EC00320
SMOVL C00321 +MOVJ EC00321
SMOVL C00322 +MOVJ EC00322
SMOVL C00323 +MOVJ EC00323
SMOVL C00324 +MOVJ EC00324
SMOVL C00325 +MOVJ EC00325
SMOVL C00326 +MOVJ EC00326
SMOVL C00327 +MOVJ EC00327
SMOVL C00328 +MOVJ EC00328
SMOVL C00329 +MOVJ EC00329
SMOVL C00330 +MOVJ EC00330
SMOVL C00331 +MOVJ EC00331
SMOVL C00332 +MOVJ EC00332
SMOVL C00333 +MOVJ EC00333
SMOVL C00334 +MOVJ EC00334
SMOVL C00335 +MOVJ EC00335
SMOVL C00336 +MOVJ EC00336
SMOVL C00337 +MOVJ EC00337
SMOVL C00338 +MOVJ EC00338
SMOVL C00339 +MOVJ EC00339
SMOVL C00340 +MOVJ EC00340
SMOVL C00341 +MOVJ EC00341
SMOVL C00342 +MOVJ EC00342
SMOVL C00343 +MOVJ EC00343
SMOVL C00344 +MOVJ EC00344
SMOVL C00345 +MOVJ EC00345
SMOVL C00346 +MOVJ EC00346
SMOVL C00347 +MOVJ EC00347
SMOVL C00348 +MOVJ EC00348
SMOVL C00349 +MOVJ EC00349
SMOVL C00350 +MOVJ EC00350
SMOVL C00351 +MOVJ EC00351
SMOVL C00352 +MOVJ EC00352
SMOVL C00353 +MOVJ EC00353
SMOVL C00354 +MOVJ EC00354
SMOVL C00355 +MOVJ EC00355
SMOVL C00356 +MOVJ EC00356
SMOVL C00357 +MOVJ EC00357
SMOVL C00358 +MOVJ EC00358
SMOVL C00359 +MOVJ EC00359
SMOVL C00360 +MOVJ EC00360
SMOVL C00361 +MOVJ EC00361
SMOVL C00362 +MOVJ EC00362
SMOVL C00363 +MOVJ EC00363
SMOVL C00364 +MOVJ EC00364
SMOVL C00365 +MOVJ EC00365
SMOVL C00366 +MOVJ EC00366
SMOVL C00367 +MOVJ EC00367
SMOVL C00368 +MOVJ EC00368
SMOVL C00369 +MOVJ EC00369
SMOVL C00370 +MOVJ EC00370
SMOVL C00371 +MOVJ EC00371
SMOVL C00372 +MOVJ EC00372
SMOVL C00373 +MOVJ EC00373
SMOVL C00374 +MOVJ EC00374
SMOVL C00375 +MOVJ EC00375
SMOVL C00376 +MOVJ EC00376
SMOVL C00377 +MOVJ EC00377
SMOVL C00378 +MOVJ EC00378
SMOVL C00379 +MOVJ EC00379
SMOVL C00380 +MOVJ EC00380
SMOVL C00381 +MOVJ EC00381
SMOVL C00382 +MOVJ EC00382
SMOVL C00383 +MOVJ EC00383
SMOVL C00384 +MOVJ EC00384
SMOVL C00385 +MOVJ EC00385
SMOVL C00386 +MOVJ EC00386
SMOVL C00387 +MOVJ EC00387
SMOVL C00388 +MOVJ EC00388
SMOVL C00389 +MOVJ EC00389
SMOVL C00390 +MOVJ EC00390
SMOVL C00391 +MOVJ EC00391
SMOVL C00392 +MOVJ EC00392
SMOVL C00393 +MOVJ EC00393
SMOVL C00394 +MOVJ EC00394
SMOVL C00395 +MOVJ EC00395
SMOVL C00396 +MOVJ EC00396
SMOVL C00397 +MOVJ EC00397
SMOVL C00398 +MOVJ EC00398
SMOVL C00399 +MOVJ EC00399
SMOVL C00400 +MOVJ EC00400
SMOVL C00401 +MOVJ EC00401
SMOVL C00402 +MOVJ EC00402
SMOVL C00403 +MOVJ EC00403
SMOVL C00404 +MOVJ EC00404
SMOVL C00405 +MOVJ EC00405
SMOVL C00406 +MOVJ EC00406
SMOVL C00407 +MOVJ EC00407
SMOVL C00408 +MOVJ EC00408
SMOVL C00409 +MOVJ EC00409
SMOVL C00410 +MOVJ EC00410
SMOVL C00411 +MOVJ EC00411
SMOVL C00412 +MOVJ EC00412
SMOVL C00413 +MOVJ EC00413
SMOVL C00414 +MOVJ EC00414
SMOVL C00415 +MOVJ EC00415
SMOVL C00416 +MOVJ EC00416
SMOVL C00417 +MOVJ EC00417
SMOVL C00418 +MOVJ EC00418
SMOVL C00419 +MOVJ EC00419
SMOVL C00420 +MOVJ EC00420
SMOVL C00421 +MOVJ EC00421
SMOVL C00422 +MOVJ EC00422
SMOVL C00423 +MOVJ EC00423
SMOVL C00424 +MOVJ EC00424
SMOVL C00425 +MOVJ EC00425
SMOVL C00426 +MOVJ EC00426
SMOVL C00427 +MOVJ EC00427
SMOVL C00428 +MOVJ EC00428
SMOVL C00429 +MOVJ EC00429
SMOVL C00430 +MOVJ EC00430
SMOVL C00431 +MOVJ EC00431
SMOVL C00432 +MOVJ EC00432
SMOVL C00433 +MOVJ EC00433
SMOVL C00434 +MOVJ EC00434
SMOVL C00435 +MOVJ EC00435
SMOVL C00436 +MOVJ EC00436
SMOVL C00437 +MOVJ EC00437
SMOVL C00438 +MOVJ EC00438
SMOVL C00439 +MOVJ EC00439
SMOVL C00440 +MOVJ EC00440
SMOVL C00441 +MOVJ EC00441
SMOVL C00442 +MOVJ EC00442
SMOVL C00443 +MOVJ EC00443
SMOVL C00444 +MOVJ EC00444
SMOVL C00445 +MOVJ EC00445
SMOVL C00446 +MOVJ EC00446
SMOVL C00447 +MOVJ EC00447
SMOVL C00448 +MOVJ EC00448
SMOVL C00449 +MOVJ EC00449
SMOVL C00450 +MOVJ EC00450
SMOVL C00451 +MOVJ EC00451
SMOVL C00452 +MOVJ EC00452
SMOVL C00453 +MOVJ EC00453
SMOVL C00454 +MOVJ EC00454
SMOVL C00455 +MOVJ EC00455
SMOVL C00456 +MOVJ EC00456
SMOVL C00457 +MOVJ EC00457
SMOVL C00458 +MOVJ EC00458
SMOVL C00459 +MOVJ EC00459
SMOVL C00460 +MOVJ EC00460
SMOVL C00461 +MOVJ EC00461
SMOVL C00462 +MOVJ EC00462
SMOVL C00463 +MOVJ EC00463
SMOVL C00464 +MOVJ EC00464
SMOVL C00465 +MOVJ EC00465
SMOVL C00466 +MOVJ EC00466
SMOVL C00467 +MOVJ EC00467
SMOVL C00468 +MOVJ EC00468
SMOVL C00469 +MOVJ EC00469
SMOVL C00470 +MOVJ EC00470
SMOVL C00471 +MOVJ EC00471
SMOVL C00472 +MOVJ EC00472
SMOVL C00473 +MOVJ EC00473
SMOVL C00474 +MOVJ EC00474
SMOVL C00475 +MOVJ EC00475
SMOVL C00476 +MOVJ EC00476
SMOVL C00477 +MOVJ EC00477
SMOVL C00478 +MOVJ EC00478
SMOVL C00479 +MOVJ EC00479
SMOVL C00480 +MOVJ EC00480
SMOVL C00481 +MOVJ EC00481
SMOVL C00482 +MOVJ EC00482
SMOVL C00483 +MOVJ EC00483
SMOVL C00484 +MOVJ EC00484
SMOVL C00485 +MOVJ EC00485
SMOVL C00486 +MOVJ EC00486
SMOVL C00487 +MOVJ EC00487
SMOVL C00488 +MOVJ EC00488
SMOVL C00489 +MOVJ EC00489
SMOVL C00490 +MOVJ EC00490
SMOVL C00491 +MOVJ EC00491
SMOVL C00492 +MOVJ EC00492
SMOVL C00493 +MOVJ EC00493
SMOVL C00494 +MOVJ EC00494
SMOVL C00495 +MOVJ EC00495
SMOVL C00496 +MOVJ EC00496
SMOVL C00497 +MOVJ EC00497
SMOVL C00498 +MOVJ EC00498
SMOVL C00499 +MOVJ EC00499
SMOVL C00500 +MOVJ EC00500
SMOVL C00501 +MOVJ EC00501
SMOVL C00502 +MOVJ EC00502
SMOVL C00503 +MOVJ EC00503
SMOVL C00504 +MOVJ EC00504
SMOVL C00505 +MOVJ EC00505
SMOVL C00506 +MOVJ EC00506
SMOVL C00507 +MOVJ EC00507
SMOVL C00508 +MOVJ EC00508
SMOVL C00509 +MOVJ EC00509
SMOVL C00510 +MOVJ EC00510
SMOVL C00511 +MOVJ EC00511
SMOVL C00512 +MOVJ EC00512
SMOVL C00513 +MOVJ EC00513
SMOVL C00514 +MOVJ EC00514
SMOVL C00515 +MOVJ EC00515
SMOVL C00516 +MOVJ EC00516
SMOVL C00517 +MOVJ EC00517
SMOVL C00518 +MOVJ EC00518
SMOVL C00519 +MOVJ EC00519
SMOVL C00520 +MOVJ EC00520
SMOVL C00521 +MOVJ EC00521
SMOVL C00522 +MOVJ EC00522
SMOVL C00523 +MOVJ EC00523
SMOVL C00524 +MOVJ EC00524
SMOVL C00525 +MOVJ EC00525
SMOVL C00526 +MOVJ EC00526
SMOVL C00527 +MOVJ EC00527
SMOVL C00528 +MOVJ EC00528
SMOVL C00529 +MOVJ EC00529
SMOVL C00530 +MOVJ EC00530
SMOVL C00531 +MOVJ EC00531
SMOVL C00532 +MOVJ EC00532
SMOVL C00533 +MOVJ EC00533
SMOVL C00534 +MOVJ EC00534
SMOVL C00535 +MOVJ EC00535
SMOVL C00536 +MOVJ EC00536
SMOVL C00537 +MOVJ EC00537
SMOVL C00538 +MOVJ EC00538
SMOVL C00539 +MOVJ EC00539
SMOVL C00540 +MOVJ EC00540
SMOVL C00541 +MOVJ EC00541
SMOVL C00542 +MOVJ EC00542
SMOVL C00543 +MOVJ EC00543
SMOVL C00544 +MOVJ EC00544
SMOVL C00545 +MOVJ EC00545
SMOVL C00546 +MOVJ EC00546
SMOVL C00547 +MOVJ EC00547
SMOVL C00548 +MOVJ EC00548
SMOVL C00549 +MOVJ EC00549
SMOVL C00550 +MOVJ EC00550
SMOVL C00551 +MOVJ EC00551
SMOVL C00552 +MOVJ EC00552
SMOVL C00553 +MOVJ EC00553
SMOVL C00554 +MOVJ EC00554
SMOVL C00555 +MOVJ EC00555
SMOVL C00556 +MOVJ EC00556
SMOVL C00557 +MOVJ EC00557
SMOVL C00558 +MOVJ EC00558
SMOVL C00559 +MOVJ EC00559
SMOVL C00560 +MOVJ EC00560
SMOVL C00561 +MOVJ EC00561
SMOVL C00562 +MOVJ EC00562
SMOVL C00563 +MOVJ EC00563
SMOVL C00564 +MOVJ EC00564
SMOVL C00565 +MOVJ EC00565
SMOVL C00566 +MOVJ EC00566
SMOVL C00567 +MOVJ EC00567
SMOVL C00568 +MOVJ EC00568
SMOVL C00569 +MOVJ EC00569
SMOVL C00570 +MOVJ EC00570
SMOVL C00571 +MOVJ EC00571
SMOVL C00572 +MOVJ EC00572
SMOVL C00573 +MOVJ EC00573
SMOVL C00574 +MOVJ EC00574
SMOVL C00575 +MOVJ EC00575
SMOVL C00576 +MOVJ EC00576
SMOVL C00577 +MOVJ EC00577
SMOVL C00578 +MOVJ EC00578
SMOVL C00579 +MOVJ EC00579
SMOVL C00580 +MOVJ EC00580
SMOVL C00581 +MOVJ EC00581
SMOVL C00582 +MOVJ EC00582
SMOVL C00583 +MOVJ EC00583
SMOVL C00584 +MOVJ EC00584
SMOVL C00585 +MOVJ EC00585
SMOVL C00586 +MOVJ EC00586
SMOVL C00587 +MOVJ EC00587
SMOVL C00588 +MOVJ EC00588
SMOVL C00589 +MOVJ EC00589
SMOVL C00590 +MOVJ EC00590
SMOVL C00591 +MOVJ EC00591
SMOVL C00592 +MOVJ EC00592
SMOVL C00593 +MOVJ EC00593
SMOVL C00594 +MOVJ EC00594
SMOVL C00595 +MOVJ EC00595
SMOVL C00596 +MOVJ EC00596
SMOVL C00597 +MOVJ EC00597
SMOVL C00598 +MOVJ EC00598
SMOVL C00599 +MOVJ EC00599
SMOVL C00600 +MOVJ EC00600
SMOVL C00601 +MOVJ EC00601
SMOVL C00602 +MOVJ EC00602
SMOVL C00603 +MOVJ EC00603
SMOVL C00604 +MOVJ EC00604
SMOVL C00605 +MOVJ EC00605
SMOVL C00606 +MOVJ EC00606
SMOVL C00607 +MOVJ EC00607
SMOVL C00608 +MOVJ EC00608
SMOVL C00609 +MOVJ EC00609
SMOVL C00610 +MOVJ EC00610
SMOVL C00611 +MOVJ EC00611
SMOVL C00612 +MOVJ EC00612
SMOVL C00613 +MOVJ EC00613
SMOVL C00614 +MOVJ EC00614
SMOVL C00615 +MOVJ EC00615
SMOVL C00616 +MOVJ EC00616
SMOVL C00617 +MOVJ EC00617
SMOVL C00618 +MOVJ EC00618
SMOVL C00619 +MOVJ EC00619
SMOVL C00620 +MOVJ EC00620
SMOVL C00621 +MOVJ EC00621
SMOVL C00622 +MOVJ EC00622
SMOVL C00623 +MOVJ EC00623
SMOVL C00624 +MOVJ EC00624
SMOVL C00625 +MOVJ EC00625
SMOVL C00626 +MOVJ EC00626
SMOVL C00627 +MOVJ EC00627
SMOVL C00628 +MOVJ EC00628
SMOVL C00629 +MOVJ EC00629
SMOVL C00630 +MOVJ EC00630
SMOVL C00631 +MOVJ EC00631
SMOVL C00632 +MOVJ EC00632
SMOVL C00633 +MOVJ EC00633
SMOVL C00634 +MOVJ EC00634
SMOVL C00635 +MOVJ EC00635
SMOVL C00636 +MOVJ EC00636
SMOVL C00637 +MOVJ EC00637
SMOVL C00638 +MOVJ EC00638
SMOVL C00639 +MOVJ EC00639
SMOVL C00640 +MOVJ EC00640
SMOVL C00641 +MOVJ EC00641
SMOVL C00642 +MOVJ EC00642
SMOVL C00643 +MOVJ EC00643
SMOVL C00644 +MOVJ EC00644
SMOVL C00645 +MOVJ EC00645
SMOVL C00646 +MOVJ EC00646
SMOVL C00647 +MOVJ EC00647
SMOVL C00648 +MOVJ EC00648
SMOVL C00649 +MOVJ EC00649
SMOVL C00650 +MOVJ EC00650
SMOVL C00651 +MOVJ EC00651
SMOVL C00652 +MOVJ EC00652
SMOVL C00653 +MOVJ EC00653
SMOVL C00654 +MOVJ EC00654
SMOVL C00655 +MOVJ EC00655
SMOVL C00656 +MOVJ EC00656
SMOVL C00657 +MOVJ EC00657
SMOVL C00658 +MOVJ EC00658
SMOVL C00659 +MOVJ EC00659
SMOVL C00660 +MOVJ EC00660
SMOVL C00661 +MOVJ EC00661
SMOVL C00662 +MOVJ EC00662
SMOVL C00663 +MOVJ EC00663
SMOVL C00664 +MOVJ EC00664
SMOVL C00665 +MOVJ EC00665
SMOVL C00666 +MOVJ EC00666
SMOVL C00667 +MOVJ EC00667
SMOVL C00668 +MOVJ EC00668
SMOVL C00669 +MOVJ EC00669
SMOVL C00670 +MOVJ EC00670
SMOVL C00671 +MOVJ EC00671
SMOVL C00672 +MOVJ EC00672
SMOVL C00673 +MOVJ EC00673
SMOVL C00674 +MOVJ EC00674
SMOVL C00675 +MOVJ EC00675
SMOVL C00676 +MOVJ EC00676
SMOVL C00677 +MOVJ EC00677
SMOVL C00678 +MOVJ EC00678
SMOVL C00679 +MOVJ EC00679
SMOVL C00680 +MOVJ EC00680
SMOVL C00681 +MOVJ EC00681
SMOVL C00682 +MOVJ EC00682
SMOVL C00683 +MOVJ EC00683
SMOVL C00684 +MOVJ EC00684
SMOVL C00685 +MOVJ EC00685
SMOVL C00686 +MOVJ EC00686
SMOVL C00687 +MOVJ EC00687
SMOVL C00688 +MOVJ EC00688
SMOVL C00689 +MOVJ EC00689
SMOVL C00690 +MOVJ EC00690
SMOVL C00691 +MOVJ EC00691
SMOVL C00692 +MOVJ EC00692
SMOVL C00693 +MOVJ EC00693
SMOVL C00694 +MOVJ EC00694
SMOVL C00695 +MOVJ EC00695
SMOVL C00696 +MOVJ EC00696
SMOVL C00697 +MOVJ EC00697
SMOVL C00698 +MOVJ EC00698
SMOVL C00699 +MOVJ EC00699
SMOVL C00700 +MOVJ EC00700
SMOVL C00701 +MOVJ EC00701
SMOVL C00702 +MOVJ EC00702
SMOVL C00703 +MOVJ EC00703
SMOVL C00704 +MOVJ EC00704
SMOVL C00705 +MOVJ EC00705
SMOVL C00706 +MOVJ EC00706
SMOVL C00707 +MOVJ EC00707
SMOVL C00708 +MOVJ EC00708
SMOVL C00709 +MOVJ EC00709
SMOVL C00710 +MOVJ EC00710
SMOVL C00711 +MOVJ EC00711
SMOVL C00712 +MOVJ EC00712
SMOVL C00713 +MOVJ EC00713
SMOVL C00714 +MOVJ EC00714
SMOVL C00715 +MOVJ EC00715
SMOVL C00716 +MOVJ EC00716
SMOVL C00717 +MOVJ EC00717
SMOVL C00718 +MOVJ EC00718
SMOVL C00719 +MOVJ EC00719
SMOVL C00720 +MOVJ EC00720
SMOVL C00721 +MOVJ EC00721
SMOVL C00722 +MOVJ EC00722
SMOVL C00723 +MOVJ EC00723
SMOVL C00724 +MOVJ EC00724
SMOVL C00725 +MOVJ EC00725
SMOVL C00726 +MOVJ EC00726
SMOVL C00727 +MOVJ EC00727
SMOVL C00728 +MOVJ EC00728
SMOVL C00729 +MOVJ EC00729
SMOVL C00730 +MOVJ EC00730
SMOVL C00731 +MOVJ EC00731
SMOVL C00732 +MOVJ EC00732
SMOVL C00733 +MOVJ EC00733
SMOVL C00734 +MOVJ EC00734
SMOVL C00735 +MOVJ EC00735
SMOVL C00736 +MOVJ EC00736
SMOVL C00737 +MOVJ EC00737
SMOVL C00738 +MOVJ EC00738
SMOVL C00739 +MOVJ EC00739
SMOVL C00740 +MOVJ EC00740
SMOVL C00741 +MOVJ EC00741
SMOVL C00742 +MOVJ EC00742
SMOVL C00743 +MOVJ EC00743
SMOVL C00744 +MOVJ EC00744
SMOVL C00745 +MOVJ EC00745
SMOVL C00746 +MOVJ EC00746
SMOVL C00747 +MOVJ EC00747
SMOVL C00748 +MOVJ EC00748
SMOVL C00749 +MOVJ EC00749
SMOVL C00750 +MOVJ EC00750
SMOVL C00751 +MOVJ EC00751
SMOVL C00752 +MOVJ EC00752
SMOVL C00753 +MOVJ EC00753
SMOVL C00754 +MOVJ EC00754
SMOVL C00755 +MOVJ EC00755
SMOVL C00756 +MOVJ EC00756
SMOVL C00757 +MOVJ EC00757
SMOVL C00758 +MOVJ EC00758
SMOVL C00759 +MOVJ EC00759
SMOVL C00760 +MOVJ EC00760
SMOVL C00761 +MOVJ EC00761
SMOVL C00762 +MOVJ EC00762
SMOVL C00763 +MOVJ EC00763
SMOVL C00764 +MOVJ EC00764
SMOVL C00765 +MOVJ EC00765
SMOVL C00766 +MOVJ EC00766
SMOVL C00767 +MOVJ EC00767
SMOVL C00768 +MOVJ EC00768
SMOVL C00769 +MOVJ EC00769
SMOVL C00770 +MOVJ EC00770
SMOVL C00771 +MOVJ EC00771
SMOVL C00772 +MOVJ EC00772
SMOVL C00773 +MOVJ EC00773
SMOVL C00774 +MOVJ EC00774
SMOVL C00775 +MOVJ EC00775
SMOVL C00776 +MOVJ EC00776
SMOVL C00777 +MOVJ EC00777
SMOVL C00778 +MOVJ EC00778
SMOVL C00779 +MOVJ EC00779
SMOVL C00780 +MOVJ EC00780
SMOVL C00781 +MOVJ EC00781
SMOVL C00782 +MOVJ EC00782
SMOVL C00783 +MOVJ EC00783
SMOVL C00784 +MOVJ EC00784
SMOVL C00785 +MOVJ EC00785
SMOVL C00786 +MOVJ EC00786
SMOVL C00787 +MOVJ EC00787
SMOVL C00788 +MOVJ EC00788
SMOVL C00789 +MOVJ EC00789
SMOVL C00790 +MOVJ EC00790
SMOVL C00791 +MOVJ EC00791
SMOVL C00792 +MOVJ EC00792
SMOVL C00793 +MOVJ EC00793
SMOVL C00794 +MOVJ EC00794
SMOVL C00795 +MOVJ EC00795
SMOVL C00796 +MOVJ EC00796
SMOVL C00797 +MOVJ EC00797
SMOVL C00798 +MOVJ EC00798
SMOVL C00799 +MOVJ EC00799
SMOVL C00800 +MOVJ EC00800
SMOVL C00801 +MOVJ EC00801
SMOVL C00802 +MOVJ EC00802
SMOVL C00803 +MOVJ EC00803
SMOVL C00804 +MOVJ EC00804
SMOVL C00805 +MOVJ EC00805
SMOVL C00806 +MOVJ EC00806
SMOVL C00807 +MOVJ EC00807
SMOVL C00808 +MOVJ EC00808
SMOVL C00809 +MOVJ EC00809
SMOVL C00810 +MOVJ EC00810
SMOVL C00811 +MOVJ EC00811
SMOVL C00812 +MOVJ EC00812
SMOVL C00813 +MOVJ EC00813
SMOVL C00814 +MOVJ EC00814
SMOVL C00815 +MOVJ EC00815
SMOVL C00816 +MOVJ EC00816
SMOVL C00817 +MOVJ EC00817
SMOVL C00818 +MOVJ EC00818
SMOVL C00819 +MOVJ EC00819
SMOVL C00820 +MOVJ EC00820
SMOVL C00821 +MOVJ EC00821
SMOVL C00822 +MOVJ EC00822
SMOVL C00823 +MOVJ EC00823
SMOVL C00824 +MOVJ EC00824
SMOVL C00825 +MOVJ EC00825
SMOVL C00826 +MOVJ EC00826
SMOVL C00827 +MOVJ EC00827
SMOVL C00828 +MOVJ EC00828
SMOVL C00829 +MOVJ EC00829
SMOVL C00830 +MOVJ EC00830
SMOVL C00831 +MOVJ EC00831
SMOVL C00832 +MOVJ EC00832
SMOVL C00833 +MOVJ EC00833
SMOVL C00834 +MOVJ EC00834
SMOVL C00835 +MOVJ EC00835
SMOVL C00836 +MOVJ EC00836
SMOVL C00837 +MOVJ EC00837
SMOVL C00838 +MOVJ EC00838
SMOVL C00839 +MOVJ EC00839
SMOVL C00840 +MOVJ EC00840
SMOVL C00841 +MOVJ EC00841
SMOVL C00842 +MOVJ EC00842
SMOVL C00843 +MOVJ EC00843
SMOVL C00844 +MOVJ EC00844
SMOVL C00845 +MOVJ EC00845
SMOVL C00846 +MOVJ EC00846
SMOVL C00847 +MOVJ EC00847
SMOVL C00848 +MOVJ EC00848
SMOVL C00849 +MOVJ EC00849
SMOVL C00850 +MOVJ EC00850
SMOVL C00851 +MOVJ EC00851
SMOVL C00852 +MOVJ EC00852
SMOVL C00853 +MOVJ EC00853
SMOVL C00854 +MOVJ EC00854
SMOVL C00855 +MOVJ EC00855
SMOVL C00856 +MOVJ EC00856
SMOVL C00857 +MOVJ EC00857
SMOVL C00858 +MOVJ EC00858
SMOVL C00859 +MOVJ EC00859
SMOVL C00860 +MOVJ EC00860
SMOVL C00861 +MOVJ EC00861
SMOVL C00862 +MOVJ EC00862
SMOVL C00863 +MOVJ EC00863
SMOVL C00864 +MOVJ EC00864
SMOVL C00865 +MOVJ EC00865
SMOVL C00866 +MOVJ EC00866
SMOVL C00867 +MOVJ EC00867
SMOVL C00868 +MOVJ EC00868
SMOVL C00869 +MOVJ EC00869
SMOVL C00870 +MOVJ EC00870
SMOVL C00871 +MOVJ EC00871
SMOVL C00872 +MOVJ EC00872
SMOVL C00873 +MOVJ EC00873
SMOVL C00874 +MOVJ EC00874
SMOVL C00875 +MOVJ EC00875
SMOVL C00876 +MOVJ EC00876
SMOVL C00877 +MOVJ EC00877
SMOVL C00878 +MOVJ EC00878
SMOVL C00879 +MOVJ EC00879
SMOVL C00880 +MOVJ EC00880
SMOVL C00881 +MOVJ EC00881
SMOVL C00882 +MOVJ EC00882
SMOVL C00883 +MOVJ EC00883
SMOVL C00884 +MOVJ EC00884
SMOVL C00885 +MOVJ EC00885
SMOVL C00886 +MOVJ EC00886
SMOVL C00887 +MOVJ EC00887
SMOVL C00888 +MOVJ EC00888
SMOVL C00889 +MOVJ EC00889
SMOVL C00890 +MOVJ EC00890
SMOVL C00891 +MOVJ EC00891
SMOVL C00892 +MOVJ EC00892
SMOVL C00893 +MOVJ EC00893
SMOVL C00894 +MOVJ EC00894
SMOVL C00895 +MOVJ EC00895
SMOVL C00896 +MOVJ EC00896
SMOVL C00897 +MOVJ EC00897
SMOVL C00898 +MOVJ EC00898
SMOVL C00899 +MOVJ EC00899
SMOVL C00900 +MOVJ EC00900
SMOVL C00901 +MOVJ EC00901
SMOVL C00902 +MOVJ EC00902
SMOVL C00903 +MOVJ EC00903
SMOVL C00904 +MOVJ EC00904
SMOVL C00905 +MOVJ EC00905
SMOVL C00906 +MOVJ EC00906
SMOVL C00907 +MOVJ EC00907
SMOVL C00908 +MOVJ EC00908
SMOVL C00909 +MOVJ EC00909
SMOVL C00910 +MOVJ EC00910
SMOVL C00911 +MOVJ EC00911
SMOVL C00912 +MOVJ EC00912
SMOVL C00913 +MOVJ EC00913
SMOVL C00914 +MOVJ EC00914
SMOVL C00915 +MOVJ EC00915
SMOVL C00916 +MOVJ EC00916
SMOVL C00917 +MOVJ EC00917
SMOVL C00918 +MOVJ EC00918
SMOVL C00919 +MOVJ EC00919
SMOVL C00920 +MOVJ EC00920
SMOVL C00921 +MOVJ EC00921
SMOVL C00922 +MOVJ EC00922
SMOVL C00923 +MOVJ EC00923
SMOVL C00924 +MOVJ EC00924
SMOVL C00925 +MOVJ EC00925
SMOVL C00926 +MOVJ EC00926
SMOVL C00927 +MOVJ EC00927
SMOVL C00928 +MOVJ EC00928
SMOVL C00929 +MOVJ EC00929
SMOVL C00930 +MOVJ EC00930
SMOVL C00931 +MOVJ EC00931
SMOVL C00932 +MOVJ EC00932
SMOVL C00933 +MOVJ EC00933
SMOVL C00934 +MOVJ EC00934
SMOVL C00935 +MOVJ EC00935
SMOVL C00936 +MOVJ EC00936
SMOVL C00937 +MOVJ EC00937
SMOVL C00938 +MOVJ EC00938
SMOVL C00939 +MOVJ EC00939
SMOVL C00940 +MOVJ EC00940
SMOVL C00941 +MOVJ EC00941
SMOVL C00942 +MOVJ EC00942
SMOVL C00943 +MOVJ EC00943
SMOVL C00944 +MOVJ EC00944
SMOVL C00945 +MOVJ EC00945
SMOVL C00946 +MOVJ EC00946
SMOVL C00947 +MOVJ EC00947
SMOVL C00948 +MOVJ EC00948
SMOVL C00949 +MOVJ EC00949
SMOVL C00950 +MOVJ EC00950
SMOVL C00951 +MOVJ EC00951
SMOVL C00952 +MOVJ EC00952
SMOVL C00953 +MOVJ EC00953
SMOVL C00954 +MOVJ EC00954
SMOVL C00955 +MOVJ EC00955
SMOVL C00956 +MOVJ EC00956
SMOVL C00957 +MOVJ EC00957
SMOVL C00958 +MOVJ EC00958
SMOVL C00959 +MOVJ EC00959
SMOVL C00960 +MOVJ EC00960
SMOVL C00961 +MOVJ EC00961
SMOVL C00962 +MOVJ EC00962
SMOVL C00963 +MOVJ EC00963
SMOVL C00964 +MOVJ EC00964
SMOVL C00965 +MOVJ EC00965
SMOVL C00966 +MOVJ EC00966
SMOVL C00967 +MOVJ EC00967
SMOVL C00968 +MOVJ EC00968
SMOVL C00969 +MOVJ EC00969
SMOVL C00970 +MOVJ EC00970
SMOVL C00971 +MOVJ EC00971
SMOVL C00972 +MOVJ EC00972
SMOVL C00973 +MOVJ EC00973
SMOVL C00974 +MOVJ EC00974
SMOVL C00975 +MOVJ EC00975
SMOVL C00976 +MOVJ EC00976
SMOVL C00977 +MOVJ EC00977
SMOVL C00978 +MOVJ EC00978
SMOVL C00979 +MOVJ EC00979
SMOVL C00980 +MOVJ EC00980
SMOVL C00981 +MOVJ EC00981
SMOVL C00982 +MOVJ EC00982
SMOVL C00983 +MOVJ EC00983
SMOVL C00984 +MOVJ EC00984
SMOVL C00985 +MOVJ EC00985
SMOVL C00986 +MOVJ EC00986
SMOVL C00987 +MOVJ EC00987
SMOVL C00988 +MOVJ EC00988
SMOVL C00989 +MOVJ EC00989
SMOVL C00990 +MOVJ EC00990
SMOVL C00991 +MOVJ EC00991
SMOVL C00992 +MOVJ EC00992
SMOVL C00993 +MOVJ EC00993
SMOVL C00994 +MOVJ EC00994
SMOVL C00995 +MOVJ EC00995
SMOVL C00996 +MOVJ EC00996
SMOVL C00997 +MOVJ EC00997
SMOVL C00998 +MOVJ EC00998
SMOVL C00999 +MOVJ EC00999
SMOVL C01000 +MOVJ EC01000
SMOVL C01001 +MOVJ EC01001
SMOVL C01002 +MOVJ EC01002
SMOVL C01003 +MOVJ EC01003
SMOVL C01004 +MOVJ EC01004
SMOVL C01005 +MOVJ EC01005
SMOVL C01006 +MOVJ EC01006
SMOVL C01007 +MOVJ EC01007
SMOVL C01008 +MOVJ EC01008
SMOVL C01009 +MOVJ EC01009
SMOVL C01010 +MOVJ EC01010
SMOVL C01011 +MOVJ EC01011
SMOVL C01012 +MOVJ EC01012
SMOVL C01013 +MOVJ EC01013
SMOVL C01014 +MOVJ EC01014
SMOVL C01015 +MOVJ EC01015
SMOVL C01016 +MOVJ EC01016
SMOVL C01017 +MOVJ EC01017
SMOVL C01018 +MOVJ EC01018
SMOVL C01019 +MOVJ EC01019
SMOVL C01020 +MOVJ EC01020
SMOVL C01021 +MOVJ EC01021
SMOVL C01022 +MOVJ EC01022
SMOVL C01023 +MOVJ EC01023
SMOVL C01024 +MOVJ EC01024
SMOVL C01025 +MOVJ EC01025
SMOVL C01026 +MOVJ EC01026
SMOVL C01027 +MOVJ EC01027
SMOVL C01028 +MOVJ EC01028
SMOVL C01029 +MOVJ EC01029
SMOVL C01030 +MOVJ EC01030
SMOVL C01031 +MOVJ EC01031
SMOVL C01032 +MOVJ EC01032
SMOVL C01033 +MOVJ EC01033
SMOVL C01034 +MOVJ EC01034
SMOVL C01035 +MOVJ EC01035
SMOVL C01036 +MOVJ EC01036
SMOVL C01037 +MOVJ EC01037
SMOVL C01038 +MOVJ EC01038
SMOVL C01039 +MOVJ EC01039
SMOVL C01040 +MOVJ EC01040
SMOVL C01041 +MOVJ EC01041
SMOVL C01042 +MOVJ EC01042
SMOVL C01043 +MOVJ EC01043
SMOVL C01044 +MOVJ EC01044
SMOVL C01045 +MOVJ EC01045
SMOVL C01046 +MOVJ EC01046
SMOVL C01047 +MOVJ EC01047
SMOVL C01048 +MOVJ EC01048
SMOVL C01049 +MOVJ EC01049
SMOVL C01050 +MOVJ EC01050
SMOVL C01051 +MOVJ EC01051
SMOVL C01052 +MOVJ EC01052
SMOVL C01053 +MOVJ EC01053
SMOVL C01054 +MOVJ EC01054
SMOVL C01055 +MOVJ EC01055
SMOVL C01056 +MOVJ EC01056
SMOVL C01057 +MOVJ EC01057
SMOVL C01058 +MOVJ EC01058
SMOVL C01059 +MOVJ EC01059
SMOVL C01060 +MOVJ EC01060
SMOVL C01061 +MOVJ EC01061
SMOVL C01062 +MOVJ EC01062
SMOVL C01063 +MOVJ EC01063
SMOVL C01064 +MOVJ EC01064
SMOVL C01065 +MOVJ EC01065
SMOVL C01066 +MOVJ EC01066
SMOVL C01067 +MOVJ EC01067
SMOVL C01068 +MOVJ EC01068
SMOVL C01069 +MOVJ EC01069
SMOVL C01070 +MOVJ EC01070
SMOVL C01071 +MOVJ EC01071
SMOVL C01072 +MOVJ EC01072
SMOVL C01073 +MOVJ EC01073
SMOVL C01074 +MOVJ EC01074
SMOVL C01075 +MOVJ EC01075
SMOVL C01076 +MOVJ EC01076
SMOVL C01077 +MOVJ EC01077
SMOVL C01078 +MOVJ EC01078
SMOVL C01079 +MOVJ EC01079
SMOVL C01080 +MOVJ EC01080
SMOVL C01081 +MOVJ EC01081
SMOVL C01082 +MOVJ EC01082
SMOVL C01083 +MOVJ EC01083
SMOVL C01084 +MOVJ EC01084
SMOVL C01085 +MOVJ EC01085
SMOVL C01086 +MOVJ EC01086
SMOVL C01087 +MOVJ EC01087
SMOVL C01088 +MOVJ EC01088
SMOVL C01089 +MOVJ EC01089
SMOVL C01090 +MOVJ EC01090
SMOVL C01091 +MOVJ EC01091
SMOVL C01092 +MOVJ EC01092
SMOVL C01093 +MOVJ EC01093
SMOVL C01094 +MOVJ EC01094
SMOVL C01095 +MOVJ EC01095
SMOVL C01096 +MOVJ EC01096
SMOVL C01097 +MOVJ EC01097
SMOVL C01098 +MOVJ EC01098
SMOVL C01099 +MOVJ EC01099
SMOVL C01100 +MOVJ EC01100
SMOVL C01101 +MOVJ EC01101
SMOVL C01102 +MOVJ EC01102
SMOVL C01103 +MOVJ EC01103
SMOVL C01104 +MOVJ EC01104
SMOVL C01105 +MOVJ EC01105
SMOVL C01106 +MOVJ EC01106
SMOVL C01107 +MOVJ EC01107
SMOVL C01108 +MOVJ EC01108
SMOVL C01109 +MOVJ EC01109
SMOVL C01110 +MOVJ EC01110
SMOVL C01111 +MOVJ EC01111
SMOVL C01112 +MOVJ EC01112
SMOVL C01113 +MOVJ EC01113
SMOVL C01114 +MOVJ EC01114
SMOVL C01115 +MOVJ EC01115
SMOVL C01116 +MOVJ EC01116
SMOVL C01117 +MOVJ EC01117
SMOVL C01118 +MOVJ EC01118
SMOVL C01119 +MOVJ EC01119
SMOVL C01120 +MOVJ EC01120
SMOVL C01121 +MOVJ EC01121
SMOVL C01122 +MOVJ EC01122
SMOVL C01123 +MOVJ EC01123
SMOVL C01124 +MOVJ EC01124
SMOVL C01125 +MOVJ EC01125
SMOVL C01126 +MOVJ EC01126
SMOVL C01127 +MOVJ EC01127
SMOVL C01128 +MOVJ EC01128
SMOVL C01129 +MOVJ EC01129
SMOVL C01130 +MOVJ EC01130
SMOVL C01131 +MOVJ EC01131
SMOVL C01132 +MOVJ EC01132
SMOVL C01133 +MOVJ EC01133
SMOVL C01134 +MOVJ EC01134
SMOVL C01135 +MOVJ EC01135
SMOVL C01136 +MOVJ EC01136
SMOVL C01137 +MOVJ EC01137
SMOVL C01138 +MOVJ EC01138
SMOVL C01139 +MOVJ EC01139
SMOVL C01140 +MOVJ EC01140
SMOVL C01141 +MOVJ EC01141
SMOVL C01142 +MOVJ EC01142
SMOVL C01143 +MOVJ EC01143
SMOVL C01144 +MOVJ EC01144
SMOVL C01145 +MOVJ EC01145
SMOVL C01146 +MOVJ EC01146
SMOVL C01147 +MOVJ EC01147
SMOVL C01148 +MOVJ EC01148
SMOVL C01149 +MOVJ EC01149
SMOVL C01150 +MOVJ EC01150
SMOVL C01151 +MOVJ EC01151
SMOVL C01152 +MOVJ EC01152
SMOVL C01153 +MOVJ EC01153
SMOVL C01154 +MOVJ EC01154
SMOVL C01155 +MOVJ EC01155
SMOVL C01156 +MOVJ EC01156
SMOVL C01157 +MOVJ EC01157
SMOVL C01158 +MOVJ EC01158
SMOVL C01159 +MOVJ EC01159
SMOVL C01160 +MOVJ EC01160
SMOVL C01161 +MOVJ EC01161
SMOVL C01162 +MOVJ EC01162
SMOVL C01163 +MOVJ EC01163
SMOVL C01164 +MOVJ EC01164
SMOVL C01165 +MOVJ EC01165
SMOVL C01166 +MOVJ EC01166
SMOVL C01167 +MOVJ EC01167
SMOVL C01168 +MOVJ EC01168
SMOVL C01169 +MOVJ EC01169
SMOVL C01170 +MOVJ EC01170
SMOVL C01171 +MOVJ EC01171
SMOVL C01172 +MOVJ EC01172
SMOVL C01173 +MOVJ EC01173
SMOVL C01174 +MOVJ EC01174
SMOVL C01175 +MOVJ EC01175
SMOVL C01176 +MOVJ EC01176
SMOVL C01177 +MOVJ EC01177
SMOVL C01178 +MOVJ EC01178
SMOVL C01179 +MOVJ EC01179
SMOVL C01180 +MOVJ EC01180
SMOVL C01181 +MOVJ EC01181
SMOVL C01182 +MOVJ EC01182
SMOVL C01183 +MOVJ EC01183
SMOVL C01184 +MOVJ EC01184
SMOVL C01185 +MOVJ EC01185
SMOVL C01186 +MOVJ EC01186
SMOVL C01187 +MOVJ EC01187
SMOVL C01188 +MOVJ EC01188
SMOVL C01189 +MOVJ EC01189
SMOVL C01190 +MOVJ EC01190
SMOVL C01191 +MOVJ EC01191
SMOVL C01192 +MOVJ EC01192
SMOVL C01193 +MOVJ EC01193
SMOVL C01194 +MOVJ EC01194
SMOVL C01195 +MOVJ EC01195
SMOVL C01196 +MOVJ EC01196
SMOVL C01197 +MOVJ EC01197
SMOVL C01198 +MOVJ EC01198
SMOVL C01199 +MOVJ EC01199
SMOVL C01200 +MOVJ EC01200
SMOVL C01201 +MOVJ EC01201
SMOVL C01202 +MOVJ EC01202
SMOVL C01203 +MOVJ EC01203
SMOVL C01204 +MOVJ EC01204
SMOVL C01205 +MOVJ EC01205
SMOVL C01206 +MOVJ EC01206
SMOVL C01207 +MOVJ EC01207
SMOVL C01208 +MOVJ EC01208
SMOVL C01209 +MOVJ EC01209
SMOVL C01210 +MOVJ EC01210
SMOVL C01211 +MOVJ EC01211
SMOVL C01212 +MOVJ EC01212
SMOVL C01213 +MOVJ EC01213
SMOVL C01214 +MOVJ EC01214
SMOVL C01215 +MOVJ EC01215
SMOVL C01216 +MOVJ EC01216
SMOVL C01217 +MOVJ EC01217
SMOVL C01218 +MOVJ EC01218
SMOVL C01219 +MOVJ EC01219
SMOVL C01220 +MOVJ EC01220
SMOVL C01221 +MOVJ EC01221
SMOVL C01222 +MOVJ EC01222
SMOVL C01223 +MOVJ EC01223
SMOVL C01224 +MOVJ EC01224
SMOVL C01225 +MOVJ EC01225
SMOVL C01226 +MOVJ EC01226
SMOVL C01227 +MOVJ EC01227
SMOVL C01228 +MOVJ EC01228
SMOVL C01229 +MOVJ EC01229
SMOVL C01230 +MOVJ EC01230
SMOVL C01231 +MOVJ EC01231
SMOVL C01232 +MOVJ EC01232
SMOVL C01233 +MOVJ EC01233
SMOVL C01234 +MOVJ EC01234
SMOVL C01235 +MOVJ EC01235
SMOVL C01236 +MOVJ EC01236
SMOVL C01237 +MOVJ EC01237
SMOVL C01238 +MOVJ EC01238
SMOVL C01239 +MOVJ EC01239
SMOVL C01240 +MOVJ EC01240
SMOVL C01241 +MOVJ EC01241
SMOVL C01242 +MOVJ EC01242
SMOVL C01243 +MOVJ EC01243
SMOVL C01244 +MOVJ EC01244
SMOVL C01245 +MOVJ EC01245
SMOVL C01246 +MOVJ EC01246
SMOVL C01247 +MOVJ EC01247
SMOVL C01248 +MOVJ EC01248
SMOVL C01249 +MOVJ EC01249
SMOVL C01250 +MOVJ EC01250
SMOVL C01251 +MOVJ EC01251
SMOVL C01252 +MOVJ EC01252
SMOVL C01253 +MOVJ EC01253
SMOVL C01254 +MOVJ EC01254
SMOVL C01255 +MOVJ EC01255
SMOVL C01256 +MOVJ EC01256
SMOVL C01257 +MOVJ EC01257
SMOVL C01258 +MOVJ EC01258
SMOVL C01259 +MOVJ EC01259
SMOVL C01260 +MOVJ EC01260
SMOVL C01261 +MOVJ EC01261
SMOVL C01262 +MOVJ EC01262
SMOVL C01263 +MOVJ EC01263
SMOVL C01264 +MOVJ EC01264
SMOVL C01265 +MOVJ EC01265
SMOVL C01266 +MOVJ EC01266
SMOVL C01267 +MOVJ EC01267
SMOVL C01268 +MOVJ EC01268
SMOVL C01269 +MOVJ EC01269
SMOVL C01270 +MOVJ EC01270
SMOVL C01271 +MOVJ EC01271
SMOVL C01272 +MOVJ EC01272
SMOVL C01273 +MOVJ EC01273
SMOVL C01274 +MOVJ EC01274
SMOVL C01275 +MOVJ EC01275
SMOVL C01276 +MOVJ EC01276
SMOVL C01277 +MOVJ EC01277
SMOVL C01278 +MOVJ EC01278
SMOVL C01279 +MOVJ EC01279
SMOVL C01280 +MOVJ EC01280
SMOVL C01281 +MOVJ EC01281
SMOVL C01282 +MOVJ EC01282
SMOVL C01283 +MOVJ EC01283
SMOVL C01284 +MOVJ EC01284
SMOVL C01285 +MOVJ EC01285
SMOVL C01286 +MOVJ EC01286
SMOVL C01287 +MOVJ EC01287
SMOVL C01288 +MOVJ EC01288
SMOVL C01289 +MOVJ EC01289
SMOVL C01290 +MOVJ EC01290
SMOVL C01291 +MOVJ EC01291
SMOVL C01292 +MOVJ EC01292
SMOVL C01293 +MOVJ EC01293
SMOVL C01294 +MOVJ EC01294
SMOVL C01295 +MOVJ EC01295
SMOVL C01296 +MOVJ EC01296
SMOVL C01297 +MOVJ EC01297
SMOVL C01298 +MOVJ EC01298
SMOVL C01299 +MOVJ EC01299
SMOVL C01300 +MOVJ EC01300
SMOVL C01301 +MOVJ EC01301
SMOVL C01302 +MOVJ EC01302
SMOVL C01303 +MOVJ EC01303
SMOVL C01304 +MOVJ EC01304
SMOVL C01305 +MOVJ EC01305
SMOVL C01306 +MOVJ EC01306
SMOVL C01307 +MOVJ EC01307
SMOVL C01308 +MOVJ EC01308
SMOVL C01309 +MOVJ EC01309
SMOVL C01310 +MOVJ EC01310
SMOVL C01311 +MOVJ EC01311
SMOVL C01312 +MOVJ EC01312
SMOVL C01313 +MOVJ EC01313
SMOVL C01314 +MOVJ EC01314
SMOVL C01315 +MOVJ EC01315
SMOVL C01316 +MOVJ EC01316
SMOVL C01317 +MOVJ EC01317
SMOVL C01318 +MOVJ EC01318
SMOVL C01319 +MOVJ EC01319
SMOVL C01320 +MOVJ EC01320
SMOVL C01321 +MOVJ EC01321
SMOVL C01322 +MOVJ EC01322
SMOVL C01323 +MOVJ EC01323
SMOVL C01324 +MOVJ EC01324
SMOVL C01325 +MOVJ EC01325
SMOVL C01326 +MOVJ EC01326
SMOVL C01327 +MOVJ EC01327
SMOVL C01328 +MOVJ EC01328
SMOVL C01329 +MOVJ EC01329
SMOVL C01330 +MOVJ EC01330
SMOVL C01331 +MOVJ EC01331
SMOVL C01332 +MOVJ EC01332
SMOVL C01333 +MOVJ EC01333
SMOVL C01334 +MOVJ EC01334
SMOVL C01335 +MOVJ EC01335
SMOVL C01336 +MOVJ EC01336
SMOVL C01337 +MOVJ EC01337
SMOVL C01338 +MOVJ EC01338
SMOVL C01339 +MOVJ EC01339
SMOVL C01340 +MOVJ EC01340
SMOVL C01341 +MOVJ EC01341
SMOVL C01342 +MOVJ EC01342
SMOVL C01343 +MOVJ EC01343
SMOVL C01344 +MOVJ EC01344
SMOVL C01345 +MOVJ EC01345
SMOVL C01346 +MOVJ EC01346
SMOVL C01347 +MOVJ EC01347
SMOVL C01348 +MOVJ EC01348
SMOVL C01349 +MOVJ EC01349
SMOVL C01350 +MOVJ EC01350
SMOVL C01351 +MOVJ EC01351
SMOVL C01352 +MOVJ EC01352
SMOVL C01353 +MOVJ EC01353
SMOVL C01354 +MOVJ EC01354
SMOVL C01355 +MOVJ EC01355
SMOVL C01356 +MOVJ EC01356
SMOVL C01357 +MOVJ EC01357
SMOVL C01358 +MOVJ EC01358
SMOVL C01359 +MOVJ EC01359
SMOVL C01360 +MOVJ EC01360
SMOVL C01361 +MOVJ EC01361
SMOVL C01362 +MOVJ EC01362
SMOVL C01363 +MOVJ EC01363
SMOVL C01364 +MOVJ EC01364
SMOVL C01365 +MOVJ EC01365
SMOVL C01366 +MOVJ EC01366
SMOVL C01367 +MOVJ EC01367
SMOVL C01368 +MOVJ EC01368
SMOVL C01369 +MOVJ EC01369
SMOVL C01370 +MOVJ EC01370
SMOVL C01371 +MOVJ EC01371
SMOVL C01372 +MOVJ EC01372
SMOVL C01373 +MOVJ EC01373
SMOVL C01374 +MOVJ EC01374
SMOVL C01375 +MOVJ EC01375
SMOVL C01376 +MOVJ EC01376
SMOVL C01377 +MOVJ EC01377
SMOVL C01378 +MOVJ EC01378
SMOVL C01379 +MOVJ EC01379
SMOVL C01380 +MOVJ EC01380
SMOVL C01381 +MOVJ EC01381
SMOVL C01382 +MOVJ EC01382
SMOVL C01383 +MOVJ EC01383
SMOVL C01384 +MOVJ EC01384
SMOVL C01385 +MOVJ EC01385
SMOVL C01386 +MOVJ EC01386
SMOVL C01387 +MOVJ EC01387
SMOVL C01388 +MOVJ EC01388
SMOVL C01389 +MOVJ EC01389
SMOVL C01390 +MOVJ EC01390
SMOVL C01391 +MOVJ EC01391
SMOVL C01392 +MOVJ EC01392
SMOVL C01393 +MOVJ EC01393
SMOVL C01394 +MOVJ EC01394
SMOVL C01395 +MOVJ EC01395
SMOVL C01396 +MOVJ EC01396
SMOVL C01397 +MOVJ EC01397
SMOVL C01398 +MOVJ EC01398
SMOVL C01399 +MOVJ EC01399
SMOVL C01400 +MOVJ EC01400
SMOVL C01401 +MOVJ EC01401
SMOVL C01402 +MOVJ EC01402
SMOVL C01403 +MOVJ EC01403
SMOVL C01404 +MOVJ EC01404
SMOVL C01405 +MOVJ EC01405
SMOVL C01406 +MOVJ EC01406
SMOVL C01407 +MOVJ EC01407
SMOVL C01408 +MOVJ EC01408
SMOVL C01409 +MOVJ EC01409
SMOVL C01410 +MOVJ EC01410
SMOVL C01411 +MOVJ EC01411
SMOVL C01412 +MOVJ EC01412
SMOVL C01413 +MOVJ EC01413
SMOVL C01414 +MOVJ EC01414
SMOVL C01415 +MOVJ EC01415
SMOVL C01416 +MOVJ EC01416
SMOVL C01417 +MOVJ EC01417
SMOVL C01418 +MOVJ EC01418
SMOVL C01419 +MOVJ EC01419
SMOVL C01420 +MOVJ EC01420
SMOVL C01421 +MOVJ EC01421
SMOVL C01422 +MOVJ EC01422
SMOVL C01423 +MOVJ EC01423
SMOVL C01424 +MOVJ EC01424
SMOVL C01425 +MOVJ EC01425
SMOVL C01426 +MOVJ EC01426
SMOVL C01427 +MOVJ EC01427
SMOVL C01428 +MOVJ EC01428
SMOVL C01429 +MOVJ EC01429
SMOVL C01430 +MOVJ EC01430
SMOVL C01431 +MOVJ EC01431
SMOVL C01432 +MOVJ EC01432
SMOVL C01433 +MOVJ EC01433
SMOVL C01434 +MOVJ EC01434
SMOVL C01435 +MOVJ EC01435
SMOVL C01436 +MOVJ EC01436
SMOVL C01437 +MOVJ EC01437
SMOVL C01438 +MOVJ EC01438
SMOVL C01439 +MOVJ EC01439
SMOVL C01440 +MOVJ EC01440
SMOVL C01441 +MOVJ EC01441
SMOVL C01442 +MOVJ EC01442
SMOVL C01443 +MOVJ EC01443
SMOVL C01444 +MOVJ EC01444
SMOVL C01445 +MOVJ EC01445
SMOVL C01446 +MOVJ EC01446
SMOVL C01447 +MOVJ EC01447
SMOVL C01448 +MOVJ EC01448
SMOVL C01449 +MOVJ EC01449
SMOVL C01450 +MOVJ EC01450
SMOVL C01451 +MOVJ EC01451
SMOVL C01452 +MOVJ EC01452
SMOVL C01453 +MOVJ EC01453
SMOVL C01454 +MOVJ EC01454
SMOVL C01455 +MOVJ EC01455
SMOVL C01456 +MOVJ EC01456
SMOVL C01457 +MOVJ EC01457
SMOVL C01458 +MOVJ EC01458
SMOVL C01459 +MOVJ EC01459
SMOVL C01460 +MOVJ EC01460
SMOVL C01461 +MOVJ EC01461
SMOVL C01462 +MOVJ EC01462
SMOVL C01463 +MOVJ EC01463
SMOVL C01464 +MOVJ EC01464
SMOVL C01465 +MOVJ EC01465
SMOVL C01466 +MOVJ EC01466
SMOVL C01467 +MOVJ EC01467
SMOVL C01468 +MOVJ EC01468
SMOVL C01469 +MOVJ EC01469
SMOVL C01470 +MOVJ EC01470
SMOVL C01471 +MOVJ EC01471
SMOVL C01472 +MOVJ EC01472
SMOVL C01473 +MOVJ EC01473
SMOVL C01474 +MOVJ EC01474
SMOVL C01475 +MOVJ EC01475
SMOVL C01476 +MOVJ EC01476
SMOVL C01477 +MOVJ EC01477
SMOVL C01478 +MOVJ EC01478
SMOVL C01479 +MOVJ EC01479
SMOVL C01480 +MOVJ EC01480
SMOVL C01481 +MOVJ EC01481
SMOVL C01482 +MOVJ EC01482
SMOVL C01483 +MOVJ EC01483
SMOVL C01484 +MOVJ EC01484
SMOVL C01485 +MOVJ EC01485
SMOVL C01486 +MOVJ EC01486
SMOVL C01487 +MOVJ EC01487
SMOVL C01488 +MOVJ EC01488
SMOVL C01489 +MOVJ EC01489
SMOVL C01490 +MOVJ EC01490
SMOVL C01491 +MOVJ EC01491
SMOVL C01492 +MOVJ EC01492
SMOVL C01493 +MOVJ EC01493
SMOVL C01494 +MOVJ EC01494
SMOVL C01495 +MOVJ EC01495
SMOVL C01496 +MOVJ EC01496
SMOVL C01497 +MOVJ EC01497
SMOVL C01498 +MOVJ EC01498
SMOVL C01499 +MOVJ EC01499
SMOVL C01500 +MOVJ EC01500
SMOVL C01501 +MOVJ EC01501
SMOVL C01502 +MOVJ EC01502
SMOVL C01503 +MOVJ EC01503
SMOVL C01504 +MOVJ EC01504
SMOVL C01505 +MOVJ EC01505
SMOVL C01506 +MOVJ EC01506
SMOVL C01507 +MOVJ EC01507
SMOVL C01508 +MOVJ EC01508
SMOVL C01509 +MOVJ EC01509
SMOVL C01510 +MOVJ EC01510
SMOVL C01511 +MOVJ EC01511
SMOVL C01512 +MOVJ EC01512
SMOVL C01513 +MOVJ EC01513
SMOVL C01514 +MOVJ EC01514
SMOVL C01515 +MOVJ EC01515
SMOVL C01516 +MOVJ EC01516
SMOVL C01517 +MOVJ EC01517
SMOVL C01518 +MOVJ EC01518
SMOVL C01519 +MOVJ EC01519
SMOVL C01520 +MOVJ EC01520
SMOVL C01521 +MOVJ EC01521
SMOVL C01522 +MOVJ EC01522
SMOVL C01523 +MOVJ EC01523
SMOVL C01524 +MOVJ EC01524
SMOVL C01525 +MOVJ EC01525
SMOVL C01526 +MOVJ EC01526
SMOVL C01527 +MOVJ EC01527
SMOVL C01528 +MOVJ EC01528
SMOVL C01529 +MOVJ EC01529
SMOVL C01530 +MOVJ EC01530
SMOVL C01531 +MOVJ EC01531
SMOVL C01532 +MOVJ EC01532
SMOVL C01533 +MOVJ EC01533
SMOVL C01534 +MOVJ EC01534
SMOVL C01535 +MOVJ EC01535
SMOVL C01536 +MOVJ EC01536
SMOVL C01537 +MOVJ EC01537
SMOVL C01538 +MOVJ EC01538
SMOVL C01539 +MOVJ EC01539
SMOVL C01540 +MOVJ EC01540
SMOVL C01541 +MOVJ EC01541
SMOVL C01542 +MOVJ EC01542
SMOVL C01543 +MOVJ EC01543
SMOVL C01544 +MOVJ EC01544
SMOVL C01545 +MOVJ EC01545
SMOVL C01546 +MOVJ EC01546
SMOVL C01547 +MOVJ EC01547
SMOVL C01548 +MOVJ EC01548
SMOVL C01549 +MOVJ EC01549
SMOVL C01550 +MOVJ EC01550
SMOVL C01551 +MOVJ EC01551
SMOVL C01552 +MOVJ EC01552
SMOVL C01553 +MOVJ EC01553
SMOVL C01554 +MOVJ EC01554
SMOVL C01555 +MOVJ EC01555
SMOVL C01556 +MOVJ EC01556
SMOVL C01557 +MOVJ EC01557
SMOVL C01558 +MOVJ EC01558
SMOVL C01559 +MOVJ EC01559
SMOVL C01560 +MOVJ EC01560
SMOVL C01561 +MOVJ EC01561
SMOVL C01562 +MOVJ EC01562
SMOVL C01563 +MOVJ EC01563
SMOVL C01564 +MOVJ EC01564
SMOVL C01565 +MOVJ EC01565
SMOVL C01566 +MOVJ EC01566
SMOVL C01567 +MOVJ EC01567
SMOVL C01568 +MOVJ EC01568
SMOVL C01569 +MOVJ EC01569
SMOVL C01570 +MOVJ EC01570
SMOVL C01571 +MOVJ EC01571
SMOVL C01572 +MOVJ EC01572
SMOVL C01573 +MOVJ EC01573
SMOVL C01574 +MOVJ EC01574
SMOVL C01575 +MOVJ EC01575
SMOVL C01576 +MOVJ EC01576
SMOVL C01577 +MOVJ EC01577
SMOVL C01578 +MOVJ EC01578
SMOVL C01579 +MOVJ EC01579
SMOVL C01580 +MOVJ EC01580
SMOVL C01581 +MOVJ EC01581
SMOVL C01582 +MOVJ EC01582
SMOVL C01583 +MOVJ EC01583
SMOVL C01584 +MOVJ EC01584
SMOVL C01585 +MOVJ EC01585
SMOVL C01586 +MOVJ EC01586
SMOVL C01587 +MOVJ EC01587
SMOVL C01588 +MOVJ EC01588
SMOVL C01589 +MOVJ EC01589
SMOVL C01590 +MOVJ EC01590
SMOVL C01591 +MOVJ EC01591
SMOVL C01592 +MOVJ EC01592
SMOVL C01593 +MOVJ EC01593
SMOVL C01594 +MOVJ EC01594
SMOVL C01595 +MOVJ EC01595
SMOVL C01596 +MOVJ EC01596
SMOVL C01597 +MOVJ EC01597
SMOVL C01598 +MOVJ EC01598
SMOVL C01599 +MOVJ EC01599
SMOVL C01600 +MOVJ EC01600
SMOVL C01601 +MOVJ EC01601
SMOVL C01602 +MOVJ EC01602
SMOVL C01603 +MOVJ EC01603
SMOVL C01604 +MOVJ EC01604
SMOVL C01605 +MOVJ EC01605
SMOVL C01606 +MOVJ EC01606
SMOVL C01607 +MOVJ EC01607
SMOVL C01608 +MOVJ EC01608
SMOVL C01609 +MOVJ EC01609
SMOVL C01610 +MOVJ EC01610
SMOVL C01611 +MOVJ EC01611
SMOVL C01612 +MOVJ EC01612
SMOVL C01613 +MOVJ EC01613
SMOVL C01614 +MOVJ EC01614
SMOVL C01615 +MOVJ EC01615
SMOVL C01616 +MOVJ EC01616
SMOVL C01617 +MOVJ EC01617
SMOVL C01618 +MOVJ EC01618
SMOVL C01619 +MOVJ EC01619
SMOVL C01620 +MOVJ EC01620
SMOVL C01621 +MOVJ EC01621
SMOVL C01622 +MOVJ EC01622
SMOVL C01623 +MOVJ EC01623
SMOVL C01624 +MOVJ EC01624
SMOVL C01625 +MOVJ EC01625
SMOVL C01626 +MOVJ EC01626
SMOVL C01627 +MOVJ EC01627
SMOVL C01628 +MOVJ EC01628
SMOVL C01629 +MOVJ EC01629
SMOVL C01630 +MOVJ EC01630
SMOVL C01631 +MOVJ EC01631
SMOVL C01632 +MOVJ EC01632
SMOVL C01633 +MOVJ EC01633
SMOVL C01634 +MOVJ EC01634
SMOVL C01635 +MOVJ EC01635
SMOVL C01636 +MOVJ EC01636
SMOVL C01637 +MOVJ EC01637
SMOVL C01638 +MOVJ EC01638
SMOVL C01639 +MOVJ EC01639
SMOVL C01640 +MOVJ EC01640
SMOVL C01641 +MOVJ EC01641
SMOVL C01642 +MOVJ EC01642
SMOVL C01643 +MOVJ EC01643
SMOVL C01644 +MOVJ EC01644
SMOVL C01645 +MOVJ EC01645
SMOVL C01646 +MOVJ EC01646
SMOVL C01647 +MOVJ EC01647
SMOVL C01648 +MOVJ EC01648
SMOVL C01649 +MOVJ EC01649
SMOVL C01650 +MOVJ EC01650
SMOVL C01651 +MOVJ EC01651
SMOVL C01652 +MOVJ EC01652
SMOVL C01653 +MOVJ EC01653
SMOVL C01654 +MOVJ EC01654
SMOVL C01655 +MOVJ EC01655
SMOVL C01656 +MOVJ EC01656
SMOVL C01657 +MOVJ EC01657
SMOVL C01658 +MOVJ EC01658
SMOVL C01659 +MOVJ EC01659
SMOVL C01660 +MOVJ EC01660
SMOVL C01661 +MOVJ EC01661
SMOVL C01662 +MOVJ EC01662
SMOVL C01663 +MOVJ EC01663
SMOVL C01664 +MOVJ EC01664
SMOVL C01665 +MOVJ EC01665
SMOVL C01666 +MOVJ EC01666
SMOVL C01667 +MOVJ EC01667
SMOVL C01668 +MOVJ EC01668
SMOVL C01669 +MOVJ EC01669
SMOVL C01670 +MOVJ EC01670
SMOVL C01671 +MOVJ EC01671
SMOVL C01672 +MOVJ EC01672
SMOVL C01673 +MOVJ EC01673
SMOVL C01674 +MOVJ EC01674
SMOVL C01675 +MOVJ EC01675
SMOVL C01676 +MOVJ EC01676
SMOVL C01677 +MOVJ EC01677
SMOVL C01678 +MOVJ EC01678
SMOVL C01679 +MOVJ EC01679
SMOVL C01680 +MOVJ EC01680
SMOVL C01681 +MOVJ EC01681
SMOVL C01682 +MOVJ EC01682
SMOVL C01683 +MOVJ EC01683
SMOVL C01684 +MOVJ EC01684
SMOVL C01685 +MOVJ EC01685
SMOVL C01686 +MOVJ EC01686
SMOVL C01687 +MOVJ EC01687
SMOVL C01688 +MOVJ EC01688
SMOVL C01689 +MOVJ EC01689
SMOVL C01690 +MOVJ EC01690
SMOVL C01691 +MOVJ EC01691
SMOVL C01692 +MOVJ EC01692
SMOVL C01693 +MOVJ EC01693
SMOVL C01694 +MOVJ EC01694
SMOVL C01695 +MOVJ EC01695
SMOVL C01696 +MOVJ EC01696
